LIN {X 0,Y 233.095,Z 584.115,A -85,B 0,C 180,E1 -19797.408,E2 -19797.408} C_VEL
LIN {X 0,Y 233.044,Z 587.862,A -85,B 0,C 180,E1 -19800,E2 -19800} C_VEL
LIN {X 0,Y 233.19,Z 589.815,A -85,B 0,C 180,E1 -19801.727,E2 -19801.727} C_VEL
LIN {X 0,Y 233.829,Z 592.542,A -85,B 0,C 180,E1 -19805.173,E2 -19805.173} C_VEL
LIN {X 0,Y 234.895,Z 593.821,A -85,B 0,C 180,E1 -19808.603,E2 -19808.603} C_VEL
LIN {X 0,Y 236.957,Z 593.579,A -85,B 0,C 180,E1 -19811.982,E2 -19811.982} C_VEL
LIN {X 0,Y 239.578,Z 591.963,A -85,B 0,C 180,E1 -19815.308,E2 -19815.308} C_VEL
LIN {X 0,Y 243.144,Z 588.902,A -85,B 0,C 180,E1 -19818.539,E2 -19818.539} C_VEL
LIN {X 0,Y 247.545,Z 584.286,A -85,B 0,C 180,E1 -19821.659,E2 -19821.659} C_VEL
LIN {X 0,Y 251.345,Z 579.836,A -85,B 0,C 180,E1 -19823.919,E2 -19823.919} C_VEL
LIN {X 0,Y 256.457,Z 573.303,A -85,B 0,C 180,E1 -19826.444,E2 -19826.444} C_VEL
LIN {X 0,Y 262.099,Z 565.298,A -85,B 0,C 180,E1 -19828.859,E2 -19828.859} C_VEL
LIN {X 0,Y 265.58,Z 559.917,A -85,B 0,C 180,E1 -19830.185,E2 -19830.185} C_VEL
LIN {X 0,Y 266.32,Z 558.434,A -85,B 0,C 180,E1 -19830.591,E2 -19830.591} C_VEL
LIN {X 0,Y 266.521,Z 553.535,A -85,B 0,C 180,E1 -19833.039,E2 -19833.039} C_VEL
LIN {X 0,Y 266.277,Z 549.635,A -85,B 0,C 180,E1 -19835.497,E2 -19835.497} C_VEL
LIN {X 0,Y 266.11,Z 548.21,A -85,B 0,C 180,E1 -19836.623,E2 -19836.623} C_VEL
LIN {X 0,Y 265.217,Z 545.882,A -85,B 0,C 180,E1 -19839.783,E2 -19839.783} C_VEL
LIN {X 0,Y 264.843,Z 545.256,A -85,B 0,C 180,E1 -19842.01,E2 -19842.01} C_VEL
LIN {X 0,Y 264.728,Z 545.601,A -85,B 0,C 180,E1 -19844.481,E2 -19844.481} C_VEL
LIN {X 0,Y 264.637,Z 546.784,A -85,B 0,C 180,E1 -19846.331,E2 -19846.331} C_VEL
LIN {X 0,Y 264.615,Z 549.004,A -85,B 0,C 180,E1 -19848.395,E2 -19848.395} C_VEL
LIN {X 0,Y 264.556,Z 552.156,A -85,B 0,C 180,E1 -19850.389,E2 -19850.389} C_VEL
LIN {X 0,Y 264.44,Z 552.98,A -85,B 0,C 180,E1 -19850.801,E2 -19850.801} C_VEL
LIN {X 0,Y 263.759,Z 555.933,A -85,B 0,C 180,E1 -19851.912,E2 -19851.912} C_VEL
LIN {X 0,Y 262.187,Z 559.644,A -85,B 0,C 180,E1 -19852.881,E2 -19852.881} C_VEL
LIN {X 0,Y 257.063,Z 569.958,A -85,B 0,C 180,E1 -19855.355,E2 -19855.355} C_VEL
LIN {X 0,Y 256.138,Z 572.23,A -85,B 0,C 180,E1 -19856.059,E2 -19856.059} C_VEL
LIN {X 0,Y 254.206,Z 577.634,A -85,B 0,C 180,E1 -19857.845,E2 -19857.845} C_VEL
LIN {X 0,Y 251.79,Z 582.561,A -85,B 0,C 180,E1 -19859.376,E2 -19859.376} C_VEL
LIN {X 0,Y 246.124,Z 591,A -85,B 0,C 180,E1 -19861.891,E2 -19861.891} C_VEL
LIN {X 0,Y 240.216,Z 598.91,A -85,B 0,C 180,E1 -19864.898,E2 -19864.898} C_VEL
LIN {X 0,Y 235.324,Z 605.22,A -85,B 0,C 180,E1 -19868.079,E2 -19868.079} C_VEL
LIN {X 0,Y 231.591,Z 610.016,A -85,B 0,C 180,E1 -19871.419,E2 -19871.419} C_VEL
LIN {X 0,Y 229.256,Z 612.702,A -85,B 0,C 180,E1 -19873.984,E2 -19873.984} C_VEL
LIN {X 0,Y 227.193,Z 615.06,A -85,B 0,C 180,E1 -19877.494,E2 -19877.494} C_VEL
LIN {X 0,Y 226.152,Z 616.049,A -85,B 0,C 180,E1 -19881.061,E2 -19881.061} C_VEL
LIN {X 0,Y 225.922,Z 615.639,A -85,B 0,C 180,E1 -19884.645,E2 -19884.645} C_VEL
LIN {X 0,Y 226.286,Z 613.75,A -85,B 0,C 180,E1 -19888.22,E2 -19888.22} C_VEL
LIN {X 0,Y 226.588,Z 612.17,A -85,B 0,C 180,E1 -19890,E2 -19890} C_VEL
LIN {X 0,Y 226.502,Z 608.882,A -85,B 0,C 180,E1 -19892.667,E2 -19892.667} C_VEL
LIN {X 0,Y 226.549,Z 604.491,A -85,B 0,C 180,E1 -19895.34,E2 -19895.34} C_VEL
LIN {X 0,Y 226.752,Z 597.802,A -85,B 0,C 180,E1 -19898.466,E2 -19898.466} C_VEL
LIN {X 0,Y 227.156,Z 590.44,A -85,B 0,C 180,E1 -19901.149,E2 -19901.149} C_VEL
LIN {X 0,Y 227.998,Z 581.33,A -85,B 0,C 180,E1 -19903.821,E2 -19903.821} C_VEL
LIN {X 0,Y 229.113,Z 571.11,A -85,B 0,C 180,E1 -19906.255,E2 -19906.255} C_VEL
LIN {X 0,Y 230.451,Z 559.72,A -85,B 0,C 180,E1 -19908.434,E2 -19908.434} C_VEL
LIN {X 0,Y 229.408,Z 548.685,A -85,B 0,C 180,E1 -19910.16,E2 -19910.16} C_VEL
LIN {X 0,Y 228.165,Z 535.293,A -85,B 0,C 180,E1 -19911.853,E2 -19911.853} C_VEL
LIN {X 0,Y 227.183,Z 521.577,A -85,B 0,C 180,E1 -19913.211,E2 -19913.211} C_VEL
LIN {X 0,Y 226.928,Z 513.581,A -85,B 0,C 180,E1 -19913.863,E2 -19913.863} C_VEL
LIN {X 0,Y 228.074,Z 506.997,A -85,B 0,C 180,E1 -19919.54,E2 -19919.54} C_VEL
LIN {X 0,Y 229.249,Z 501.672,A -85,B 0,C 180,E1 -19924.134,E2 -19924.134} C_VEL
LIN {X 0,Y 229.836,Z 499.05,A -85,B 0,C 180,E1 -19926.414,E2 -19926.414} C_VEL
LIN {X 0,Y 229.367,Z 495.015,A -85,B 0,C 180,E1 -19930.05,E2 -19930.05} C_VEL
LIN {X 0,Y 228.375,Z 489.834,A -85,B 0,C 180,E1 -19934.944,E2 -19934.944} C_VEL
LIN {X 0,Y 228.135,Z 488.069,A -85,B 0,C 180,E1 -19936.73,E2 -19936.73} C_VEL
LIN {X 0,Y 227.881,Z 488.095,A -85,B 0,C 180,E1 -19941.916,E2 -19941.916} C_VEL
LIN {X 0,Y 227.891,Z 488.098,A -85,B 0,C 180,E1 -19946.373,E2 -19946.373} C_VEL
LIN {X 0,Y 227.905,Z 488.095,A -85,B 0,C 180,E1 -19950.436,E2 -19950.436} C_VEL
LIN {X 0,Y 227.929,Z 488.093,A -85,B 0,C 180,E1 -19954.426,E2 -19954.426} C_VEL
LIN {X 0,Y 227.963,Z 488.088,A -85,B 0,C 180,E1 -19958.287,E2 -19958.287} C_VEL
LIN {X 0,Y 228.036,Z 488.08,A -85,B 0,C 180,E1 -19962.826,E2 -19962.826} C_VEL
LIN {X 0,Y 228.095,Z 488.069,A -85,B 0,C 180,E1 -19967.545,E2 -19967.545} C_VEL
LIN {X 0,Y 228.327,Z 488.042,A -85,B 0,C 180,E1 -19971.147,E2 -19971.147} C_VEL
LIN {X 0,Y 228.36,Z 488.039,A -85,B 0,C 180,E1 -19972.929,E2 -19972.929} C_VEL
LIN {X 0,Y 228.556,Z 488.012,A -85,B 0,C 180,E1 -19978.238,E2 -19978.238} C_VEL
LIN {X 0,Y 228.557,Z 488.013,A -85,B 0,C 180,E1 -19981.762,E2 -19981.762} C_VEL
LIN {X 0,Y 228.36,Z 488.036,A -85,B 0,C 180,E1 -19987.072,E2 -19987.072} C_VEL
LIN {X 0,Y 228.173,Z 488.063,A -85,B 0,C 180,E1 -19990.65,E2 -19990.65} C_VEL
LIN {X 0,Y 228.06,Z 488.073,A -85,B 0,C 180,E1 -19996.102,E2 -19996.102} C_VEL
LIN {X 0,Y 227.945,Z 488.09,A -85,B 0,C 180,E1 -19999.826,E2 -19999.826} C_VEL
LIN {X 0,Y 227.916,Z 488.091,A -85,B 0,C 180,E1 -20003.633,E2 -20003.633} C_VEL
LIN {X 0,Y 227.888,Z 488.096,A -85,B 0,C 180,E1 -20007.555,E2 -20007.555} C_VEL
LIN {X 0,Y 227.874,Z 488.097,A -85,B 0,C 180,E1 -20011.622,E2 -20011.622} C_VEL
LIN {X 0,Y 227.885,Z 488.097,A -85,B 0,C 180,E1 -20015.872,E2 -20015.872} C_VEL
LIN {X 0,Y 227.827,Z 488.104,A -85,B 0,C 180,E1 -20020.377,E2 -20020.377} C_VEL
LIN {X 0,Y 227.835,Z 488.103,A -85,B 0,C 180,E1 -20025.193,E2 -20025.193} C_VEL
LIN {X 0,Y 227.835,Z 488.102,A -85,B 0,C 180,E1 -20029.625,E2 -20029.625} C_VEL
LIN {X 0,Y 227.903,Z 488.098,A -85,B 0,C 180,E1 -20034.132,E2 -20034.132} C_VEL
LIN {X 0,Y 227.875,Z 488.097,A -85,B 0,C 180,E1 -20038.379,E2 -20038.379} C_VEL
LIN {X 0,Y 227.888,Z 488.098,A -85,B 0,C 180,E1 -20042.445,E2 -20042.445} C_VEL
LIN {X 0,Y 227.917,Z 488.093,A -85,B 0,C 180,E1 -20046.368,E2 -20046.368} C_VEL
LIN {X 0,Y 227.946,Z 488.092,A -85,B 0,C 180,E1 -20050.175,E2 -20050.175} C_VEL
LIN {X 0,Y 228.061,Z 488.077,A -85,B 0,C 180,E1 -20053.898,E2 -20053.898} C_VEL
LIN {X 0,Y 228.076,Z 488.07,A -85,B 0,C 180,E1 -20057.544,E2 -20057.544} C_VEL
LIN {X 0,Y 228.263,Z 488.05,A -85,B 0,C 180,E1 -20061.145,E2 -20061.145} C_VEL
LIN {X 0,Y 228.315,Z 488.042,A -85,B 0,C 180,E1 -20062.928,E2 -20062.928} C_VEL
LIN {X 0,Y 228.558,Z 488.015,A -85,B 0,C 180,E1 -20068.238,E2 -20068.238} C_VEL
LIN {X 0,Y 228.558,Z 488.015,A -85,B 0,C 180,E1 -20071.762,E2 -20071.762} C_VEL
LIN {X 0,Y 228.328,Z 488.041,A -85,B 0,C 180,E1 -20077.072,E2 -20077.072} C_VEL
LIN {X 0,Y 228.15,Z 488.063,A -85,B 0,C 180,E1 -20080.651,E2 -20080.651} C_VEL
LIN {X 0,Y 228.069,Z 488.074,A -85,B 0,C 180,E1 -20084.272,E2 -20084.272} C_VEL
LIN {X 0,Y 228.007,Z 488.085,A -85,B 0,C 180,E1 -20087.953,E2 -20087.953} C_VEL
LIN {X 0,Y 227.934,Z 488.089,A -85,B 0,C 180,E1 -20092.329,E2 -20092.329} C_VEL
LIN {X 0,Y 227.946,Z 488.089,A -85,B 0,C 180,E1 -20096.603,E2 -20096.603} C_VEL
LIN {X 0,Y 227.911,Z 488.091,A -85,B 0,C 180,E1 -20100.296,E2 -20100.296} C_VEL
LIN {X 0,Y 227.892,Z 488.098,A -85,B 0,C 180,E1 -20103.718,E2 -20103.718} C_VEL
LIN {X 0,Y 227.873,Z 488.098,A -85,B 0,C 180,E1 -20108.086,E2 -20108.086} C_VEL
LIN {X 0,Y 227.817,Z 488.105,A -85,B 0,C 180,E1 -20112.741,E2 -20112.741} C_VEL
LIN {X 0,Y 227.812,Z 488.105,A -85,B 0,C 180,E1 -20117.257,E2 -20117.257} C_VEL
LIN {X 0,Y 227.786,Z 488.112,A -85,B 0,C 180,E1 -20121.897,E2 -20121.897} C_VEL
LIN {X 0,Y 227.697,Z 488.121,A -85,B 0,C 180,E1 -20124.094,E2 -20124.094} C_VEL
LIN {X 0,Y 227.316,Z 488.167,A -85,B 0,C 180,E1 -20128.291,E2 -20128.291} C_VEL
LIN {X 0,Y 226.929,Z 488.222,A -85,B 0,C 180,E1 -20132.318,E2 -20132.318} C_VEL
LIN {X 0,Y 226.517,Z 488.272,A -85,B 0,C 180,E1 -20136.502,E2 -20136.502} C_VEL
LIN {X 0,Y 229.096,Z 503.824,A -85,B 0,C 180,E1 -20137.96,E2 -20137.96} C_VEL
LIN {X 0,Y 231.348,Z 516.521,A -85,B 0,C 180,E1 -20139.475,E2 -20139.475} C_VEL
LIN {X 0,Y 232.042,Z 520.942,A -85,B 0,C 180,E1 -20140.077,E2 -20140.077} C_VEL
LIN {X 0,Y 230.695,Z 533.731,A -85,B 0,C 180,E1 -20142.034,E2 -20142.034} C_VEL
LIN {X 0,Y 229.335,Z 545.229,A -85,B 0,C 180,E1 -20144.218,E2 -20144.218} C_VEL
LIN {X 0,Y 228.115,Z 555.573,A -85,B 0,C 180,E1 -20146.64,E2 -20146.64} C_VEL
LIN {X 0,Y 227.179,Z 564.818,A -85,B 0,C 180,E1 -20149.303,E2 -20149.303} C_VEL
LIN {X 0,Y 226.466,Z 573.528,A -85,B 0,C 180,E1 -20152.421,E2 -20152.421} C_VEL
LIN {X 0,Y 226.079,Z 580.412,A -85,B 0,C 180,E1 -20155.542,E2 -20155.542} C_VEL
LIN {X 0,Y 225.985,Z 585.073,A -85,B 0,C 180,E1 -20158.218,E2 -20158.218} C_VEL
LIN {X 0,Y 226.119,Z 589.684,A -85,B 0,C 180,E1 -20161.781,E2 -20161.781} C_VEL
LIN {X 0,Y 226.405,Z 591.403,A -85,B 0,C 180,E1 -20163.559,E2 -20163.559} C_VEL
LIN {X 0,Y 227.226,Z 593.653,A -85,B 0,C 180,E1 -20167.106,E2 -20167.106} C_VEL
LIN {X 0,Y 228.857,Z 594.476,A -85,B 0,C 180,E1 -20170.617,E2 -20170.617} C_VEL
LIN {X 0,Y 231.32,Z 593.867,A -85,B 0,C 180,E1 -20174.067,E2 -20174.067} C_VEL
LIN {X 0,Y 234.616,Z 591.845,A -85,B 0,C 180,E1 -20177.431,E2 -20177.431} C_VEL
LIN {X 0,Y 238.783,Z 588.417,A -85,B 0,C 180,E1 -20180.682,E2 -20180.682} C_VEL
LIN {X 0,Y 243.747,Z 583.472,A -85,B 0,C 180,E1 -20183.807,E2 -20183.807} C_VEL
LIN {X 0,Y 249.667,Z 576.905,A -85,B 0,C 180,E1 -20186.769,E2 -20186.769} C_VEL
LIN {X 0,Y 256.354,Z 568.409,A -85,B 0,C 180,E1 -20189.569,E2 -20189.569} C_VEL
LIN {X 0,Y 259.937,Z 563.469,A -85,B 0,C 180,E1 -20190.911,E2 -20190.911} C_VEL
LIN {X 0,Y 261.012,Z 561.597,A -85,B 0,C 180,E1 -20191.474,E2 -20191.474} C_VEL
LIN {X 0,Y 261.39,Z 557.918,A -85,B 0,C 180,E1 -20193.54,E2 -20193.54} C_VEL
LIN {X 0,Y 261.426,Z 554.117,A -85,B 0,C 180,E1 -20196.244,E2 -20196.244} C_VEL
LIN {X 0,Y 260.976,Z 552.102,A -85,B 0,C 180,E1 -20198.651,E2 -20198.651} C_VEL
LIN {X 0,Y 260.607,Z 551.108,A -85,B 0,C 180,E1 -20200.965,E2 -20200.965} C_VEL
LIN {X 0,Y 260.477,Z 550.912,A -85,B 0,C 180,E1 -20203.239,E2 -20203.239} C_VEL
LIN {X 0,Y 260.343,Z 551.8,A -85,B 0,C 180,E1 -20205.422,E2 -20205.422} C_VEL
LIN {X 0,Y 260.165,Z 553.684,A -85,B 0,C 180,E1 -20207.519,E2 -20207.519} C_VEL
LIN {X 0,Y 259.949,Z 556.429,A -85,B 0,C 180,E1 -20209.544,E2 -20209.544} C_VEL
LIN {X 0,Y 259.251,Z 560.111,A -85,B 0,C 180,E1 -20211.427,E2 -20211.427} C_VEL
LIN {X 0,Y 257.672,Z 566.9,A -85,B 0,C 180,E1 -20214.152,E2 -20214.152} C_VEL
LIN {X 0,Y 256.138,Z 572.23,A -85,B 0,C 180,E1 -20216.059,E2 -20216.059} C_VEL
LIN {X 0,Y 255.085,Z 574.558,A -85,B 0,C 180,E1 -20216.743,E2 -20216.743} C_VEL
LIN {X 0,Y 253.54,Z 577.077,A -85,B 0,C 180,E1 -20217.348,E2 -20217.348} C_VEL
LIN {X 0,Y 249.505,Z 582.161,A -85,B 0,C 180,E1 -20218.416,E2 -20218.416} C_VEL
LIN {X 0,Y 242.787,Z 589.348,A -85,B 0,C 180,E1 -20220.062,E2 -20220.062} C_VEL
LIN {X 0,Y 240.884,Z 591.498,A -85,B 0,C 180,E1 -20220.727,E2 -20220.727} C_VEL
LIN {X 0,Y 235.306,Z 598.328,A -85,B 0,C 180,E1 -20223.383,E2 -20223.383} C_VEL
LIN {X 0,Y 229.312,Z 605.282,A -85,B 0,C 180,E1 -20227.027,E2 -20227.027} C_VEL
LIN {X 0,Y 225.718,Z 609.319,A -85,B 0,C 180,E1 -20229.971,E2 -20229.971} C_VEL
LIN {X 0,Y 222.436,Z 612.714,A -85,B 0,C 180,E1 -20233.479,E2 -20233.479} C_VEL
LIN {X 0,Y 220.225,Z 614.779,A -85,B 0,C 180,E1 -20237.092,E2 -20237.092} C_VEL
LIN {X 0,Y 219.122,Z 615.507,A -85,B 0,C 180,E1 -20240.772,E2 -20240.772} C_VEL
LIN {X 0,Y 218.886,Z 614.813,A -85,B 0,C 180,E1 -20244.472,E2 -20244.472} C_VEL
LIN {X 0,Y 219.274,Z 612.657,A -85,B 0,C 180,E1 -20248.163,E2 -20248.163} C_VEL
LIN {X 0,Y 219.571,Z 610.998,A -85,B 0,C 180,E1 -20250,E2 -20250} C_VEL
LIN {X 0,Y 219.498,Z 607.509,A -85,B 0,C 180,E1 -20252.753,E2 -20252.753} C_VEL
LIN {X 0,Y 219.557,Z 602.876,A -85,B 0,C 180,E1 -20255.51,E2 -20255.51} C_VEL
LIN {X 0,Y 219.734,Z 596.979,A -85,B 0,C 180,E1 -20258.275,E2 -20258.275} C_VEL
LIN {X 0,Y 220.121,Z 589.583,A -85,B 0,C 180,E1 -20261.044,E2 -20261.044} C_VEL
LIN {X 0,Y 220.962,Z 580.515,A -85,B 0,C 180,E1 -20263.801,E2 -20263.801} C_VEL
LIN {X 0,Y 221.952,Z 571.302,A -85,B 0,C 180,E1 -20266.085,E2 -20266.085} C_VEL
LIN {X 0,Y 223.289,Z 560.005,A -85,B 0,C 180,E1 -20268.346,E2 -20268.346} C_VEL
LIN {X 0,Y 222.297,Z 548.841,A -85,B 0,C 180,E1 -20270.17,E2 -20270.17} C_VEL
LIN {X 0,Y 221.092,Z 535.554,A -85,B 0,C 180,E1 -20271.932,E2 -20271.932} C_VEL
LIN {X 0,Y 220.099,Z 521.557,A -85,B 0,C 180,E1 -20273.386,E2 -20273.386} C_VEL
LIN {X 0,Y 219.834,Z 513.247,A -85,B 0,C 180,E1 -20274.054,E2 -20274.054} C_VEL
LIN {X 0,Y 220.969,Z 507.128,A -85,B 0,C 180,E1 -20279.537,E2 -20279.537} C_VEL
LIN {X 0,Y 222.295,Z 501.353,A -85,B 0,C 180,E1 -20284.714,E2 -20284.714} C_VEL
LIN {X 0,Y 222.721,Z 498.997,A -85,B 0,C 180,E1 -20286.837,E2 -20286.837} C_VEL
LIN {X 0,Y 222.163,Z 495.001,A -85,B 0,C 180,E1 -20290.604,E2 -20290.604} C_VEL
LIN {X 0,Y 221.201,Z 489.839,A -85,B 0,C 180,E1 -20295.655,E2 -20295.655} C_VEL
LIN {X 0,Y 221.104,Z 488.945,A -85,B 0,C 180,E1 -20296.774,E2 -20296.774} C_VEL
LIN {X 0,Y 220.866,Z 488.973,A -85,B 0,C 180,E1 -20300.476,E2 -20300.476} C_VEL
LIN {X 0,Y 220.816,Z 488.979,A -85,B 0,C 180,E1 -20305.048,E2 -20305.048} C_VEL
LIN {X 0,Y 220.834,Z 488.974,A -85,B 0,C 180,E1 -20309.39,E2 -20309.39} C_VEL
LIN {X 0,Y 220.895,Z 488.966,A -85,B 0,C 180,E1 -20313.55,E2 -20313.55} C_VEL
LIN {X 0,Y 220.879,Z 488.969,A -85,B 0,C 180,E1 -20317.554,E2 -20317.554} C_VEL
LIN {X 0,Y 220.985,Z 488.958,A -85,B 0,C 180,E1 -20322.571,E2 -20322.571} C_VEL
LIN {X 0,Y 221.028,Z 488.95,A -85,B 0,C 180,E1 -20327.14,E2 -20327.14} C_VEL
LIN {X 0,Y 221.26,Z 488.923,A -85,B 0,C 180,E1 -20330.862,E2 -20330.862} C_VEL
LIN {X 0,Y 221.313,Z 488.918,A -85,B 0,C 180,E1 -20332.703,E2 -20332.703} C_VEL
LIN {X 0,Y 221.514,Z 488.889,A -85,B 0,C 180,E1 -20338.182,E2 -20338.182} C_VEL
LIN {X 0,Y 221.515,Z 488.891,A -85,B 0,C 180,E1 -20341.818,E2 -20341.818} C_VEL
LIN {X 0,Y 221.313,Z 488.913,A -85,B 0,C 180,E1 -20347.298,E2 -20347.298} C_VEL
LIN {X 0,Y 221.119,Z 488.94,A -85,B 0,C 180,E1 -20350.994,E2 -20350.994} C_VEL
LIN {X 0,Y 221.018,Z 488.953,A -85,B 0,C 180,E1 -20356.63,E2 -20356.63} C_VEL
LIN {X 0,Y 220.895,Z 488.97,A -85,B 0,C 180,E1 -20360.486,E2 -20360.486} C_VEL
LIN {X 0,Y 220.869,Z 488.971,A -85,B 0,C 180,E1 -20364.435,E2 -20364.435} C_VEL
LIN {X 0,Y 220.839,Z 488.977,A -85,B 0,C 180,E1 -20368.514,E2 -20368.514} C_VEL
LIN {X 0,Y 220.822,Z 488.974,A -85,B 0,C 180,E1 -20372.756,E2 -20372.756} C_VEL
LIN {X 0,Y 220.813,Z 488.978,A -85,B 0,C 180,E1 -20377.279,E2 -20377.279} C_VEL
LIN {X 0,Y 220.772,Z 488.981,A -85,B 0,C 180,E1 -20381.953,E2 -20381.953} C_VEL
LIN {X 0,Y 220.776,Z 488.982,A -85,B 0,C 180,E1 -20385.547,E2 -20385.547} C_VEL
LIN {X 0,Y 220.812,Z 488.977,A -85,B 0,C 180,E1 -20390.464,E2 -20390.464} C_VEL
LIN {X 0,Y 220.834,Z 488.975,A -85,B 0,C 180,E1 -20392.795,E2 -20392.795} C_VEL
LIN {X 0,Y 220.827,Z 488.975,A -85,B 0,C 180,E1 -20397.246,E2 -20397.246} C_VEL
LIN {X 0,Y 220.839,Z 488.974,A -85,B 0,C 180,E1 -20401.487,E2 -20401.487} C_VEL
LIN {X 0,Y 220.87,Z 488.971,A -85,B 0,C 180,E1 -20405.566,E2 -20405.566} C_VEL
LIN {X 0,Y 220.896,Z 488.966,A -85,B 0,C 180,E1 -20409.514,E2 -20409.514} C_VEL
LIN {X 0,Y 221.02,Z 488.952,A -85,B 0,C 180,E1 -20413.371,E2 -20413.371} C_VEL
LIN {X 0,Y 221.085,Z 488.943,A -85,B 0,C 180,E1 -20419.005,E2 -20419.005} C_VEL
LIN {X 0,Y 221.252,Z 488.923,A -85,B 0,C 180,E1 -20422.701,E2 -20422.701} C_VEL
LIN {X 0,Y 221.515,Z 488.893,A -85,B 0,C 180,E1 -20428.182,E2 -20428.182} C_VEL
LIN {X 0,Y 221.516,Z 488.893,A -85,B 0,C 180,E1 -20431.818,E2 -20431.818} C_VEL
LIN {X 0,Y 221.263,Z 488.921,A -85,B 0,C 180,E1 -20437.3,E2 -20437.3} C_VEL
LIN {X 0,Y 221.086,Z 488.943,A -85,B 0,C 180,E1 -20440.996,E2 -20440.996} C_VEL
LIN {X 0,Y 221.021,Z 488.952,A -85,B 0,C 180,E1 -20446.63,E2 -20446.63} C_VEL
LIN {X 0,Y 220.897,Z 488.966,A -85,B 0,C 180,E1 -20450.486,E2 -20450.486} C_VEL
LIN {X 0,Y 220.871,Z 488.971,A -85,B 0,C 180,E1 -20454.435,E2 -20454.435} C_VEL
LIN {X 0,Y 220.84,Z 488.973,A -85,B 0,C 180,E1 -20458.513,E2 -20458.513} C_VEL
LIN {X 0,Y 220.827,Z 488.975,A -85,B 0,C 180,E1 -20462.755,E2 -20462.755} C_VEL
LIN {X 0,Y 220.842,Z 488.974,A -85,B 0,C 180,E1 -20467.288,E2 -20467.288} C_VEL
LIN {X 0,Y 220.778,Z 488.984,A -85,B 0,C 180,E1 -20471.951,E2 -20471.951} C_VEL
LIN {X 0,Y 220.776,Z 488.985,A -85,B 0,C 180,E1 -20475.546,E2 -20475.546} C_VEL
LIN {X 0,Y 220.771,Z 488.982,A -85,B 0,C 180,E1 -20480.455,E2 -20480.455} C_VEL
LIN {X 0,Y 220.718,Z 488.99,A -85,B 0,C 180,E1 -20482.771,E2 -20482.771} C_VEL
LIN {X 0,Y 220.364,Z 489.031,A -85,B 0,C 180,E1 -20487.167,E2 -20487.167} C_VEL
LIN {X 0,Y 219.979,Z 489.083,A -85,B 0,C 180,E1 -20491.365,E2 -20491.365} C_VEL
LIN {X 0,Y 219.534,Z 489.276,A -85,B 0,C 180,E1 -20496.349,E2 -20496.349} C_VEL
LIN {X 0,Y 221.785,Z 503.009,A -85,B 0,C 180,E1 -20497.65,E2 -20497.65} C_VEL
LIN {X 0,Y 224.089,Z 516.032,A -85,B 0,C 180,E1 -20499.22,E2 -20499.22} C_VEL
LIN {X 0,Y 224.938,Z 520.869,A -85,B 0,C 180,E1 -20499.898,E2 -20499.898} C_VEL
LIN {X 0,Y 223.614,Z 533.665,A -85,B 0,C 180,E1 -20501.918,E2 -20501.918} C_VEL
LIN {X 0,Y 222.223,Z 545.155,A -85,B 0,C 180,E1 -20504.17,E2 -20504.17} C_VEL
LIN {X 0,Y 221.006,Z 555.514,A -85,B 0,C 180,E1 -20506.67,E2 -20506.67} C_VEL
LIN {X 0,Y 220.071,Z 564.873,A -85,B 0,C 180,E1 -20509.419,E2 -20509.419} C_VEL
LIN {X 0,Y 219.346,Z 573.658,A -85,B 0,C 180,E1 -20512.636,E2 -20512.636} C_VEL
LIN {X 0,Y 219.007,Z 579.696,A -85,B 0,C 180,E1 -20515.398,E2 -20515.398} C_VEL
LIN {X 0,Y 218.919,Z 584.567,A -85,B 0,C 180,E1 -20518.16,E2 -20518.16} C_VEL
LIN {X 0,Y 218.945,Z 588.414,A -85,B 0,C 180,E1 -20520.919,E2 -20520.919} C_VEL
LIN {X 0,Y 219.346,Z 591.333,A -85,B 0,C 180,E1 -20523.674,E2 -20523.674} C_VEL
LIN {X 0,Y 220.182,Z 593.907,A -85,B 0,C 180,E1 -20527.335,E2 -20527.335} C_VEL
LIN {X 0,Y 221.913,Z 595.009,A -85,B 0,C 180,E1 -20530.954,E2 -20530.954} C_VEL
LIN {X 0,Y 224.511,Z 594.714,A -85,B 0,C 180,E1 -20534.503,E2 -20534.503} C_VEL
LIN {X 0,Y 227.955,Z 593.059,A -85,B 0,C 180,E1 -20537.957,E2 -20537.957} C_VEL
LIN {X 0,Y 232.315,Z 589.99,A -85,B 0,C 180,E1 -20541.286,E2 -20541.286} C_VEL
LIN {X 0,Y 237.53,Z 585.478,A -85,B 0,C 180,E1 -20544.471,E2 -20544.471} C_VEL
LIN {X 0,Y 242.051,Z 581.058,A -85,B 0,C 180,E1 -20546.746,E2 -20546.746} C_VEL
LIN {X 0,Y 248.862,Z 573.648,A -85,B 0,C 180,E1 -20549.618,E2 -20549.618} C_VEL
LIN {X 0,Y 255.215,Z 565.676,A -85,B 0,C 180,E1 -20552.002,E2 -20552.002} C_VEL
LIN {X 0,Y 255.674,Z 564.787,A -85,B 0,C 180,E1 -20552.393,E2 -20552.393} C_VEL
LIN {X 0,Y 256.29,Z 560.636,A -85,B 0,C 180,E1 -20555.16,E2 -20555.16} C_VEL
LIN {X 0,Y 256.446,Z 559.334,A -85,B 0,C 180,E1 -20556.23,E2 -20556.23} C_VEL
LIN {X 0,Y 256.152,Z 557.161,A -85,B 0,C 180,E1 -20559.127,E2 -20559.127} C_VEL
LIN {X 0,Y 255.896,Z 556.341,A -85,B 0,C 180,E1 -20562.137,E2 -20562.137} C_VEL
LIN {X 0,Y 255.815,Z 556.712,A -85,B 0,C 180,E1 -20564.414,E2 -20564.414} C_VEL
LIN {X 0,Y 255.553,Z 558.206,A -85,B 0,C 180,E1 -20566.565,E2 -20566.565} C_VEL
LIN {X 0,Y 255.244,Z 560.565,A -85,B 0,C 180,E1 -20568.637,E2 -20568.637} C_VEL
LIN {X 0,Y 254.383,Z 564.117,A -85,B 0,C 180,E1 -20570.676,E2 -20570.676} C_VEL
LIN {X 0,Y 252.559,Z 570.004,A -85,B 0,C 180,E1 -20573.254,E2 -20573.254} C_VEL
LIN {X 0,Y 250.113,Z 576.663,A -85,B 0,C 180,E1 -20575.806,E2 -20575.806} C_VEL
LIN {X 0,Y 247.423,Z 582.413,A -85,B 0,C 180,E1 -20577.819,E2 -20577.819} C_VEL
LIN {X 0,Y 244.311,Z 587.131,A -85,B 0,C 180,E1 -20579.295,E2 -20579.295} C_VEL
LIN {X 0,Y 240.884,Z 591.498,A -85,B 0,C 180,E1 -20580.727,E2 -20580.727} C_VEL
LIN {X 0,Y 237.881,Z 594.617,A -85,B 0,C 180,E1 -20581.71,E2 -20581.71} C_VEL
LIN {X 0,Y 231.696,Z 599.436,A -85,B 0,C 180,E1 -20583.21,E2 -20583.21} C_VEL
LIN {X 0,Y 225.744,Z 603.53,A -85,B 0,C 180,E1 -20584.876,E2 -20584.876} C_VEL
LIN {X 0,Y 223.156,Z 605.615,A -85,B 0,C 180,E1 -20586.101,E2 -20586.101} C_VEL
LIN {X 0,Y 219.064,Z 609.662,A -85,B 0,C 180,E1 -20589.335,E2 -20589.335} C_VEL
LIN {X 0,Y 215.637,Z 612.711,A -85,B 0,C 180,E1 -20592.943,E2 -20592.943} C_VEL
LIN {X 0,Y 213.273,Z 614.435,A -85,B 0,C 180,E1 -20596.663,E2 -20596.663} C_VEL
LIN {X 0,Y 212.11,Z 614.85,A -85,B 0,C 180,E1 -20600.464,E2 -20600.464} C_VEL
LIN {X 0,Y 211.851,Z 613.876,A -85,B 0,C 180,E1 -20604.401,E2 -20604.401} C_VEL
LIN {X 0,Y 212.259,Z 611.533,A -85,B 0,C 180,E1 -20608.102,E2 -20608.102} C_VEL
LIN {X 0,Y 212.573,Z 608.615,A -85,B 0,C 180,E1 -20610.947,E2 -20610.947} C_VEL
LIN {X 0,Y 212.531,Z 604.553,A -85,B 0,C 180,E1 -20613.792,E2 -20613.792} C_VEL
LIN {X 0,Y 212.622,Z 599.223,A -85,B 0,C 180,E1 -20616.68,E2 -20616.68} C_VEL
LIN {X 0,Y 212.869,Z 592.598,A -85,B 0,C 180,E1 -20619.502,E2 -20619.502} C_VEL
LIN {X 0,Y 213.534,Z 584.346,A -85,B 0,C 180,E1 -20622.353,E2 -20622.353} C_VEL
LIN {X 0,Y 214.326,Z 576.01,A -85,B 0,C 180,E1 -20624.722,E2 -20624.722} C_VEL
LIN {X 0,Y 215.422,Z 566.005,A -85,B 0,C 180,E1 -20627.075,E2 -20627.075} C_VEL
LIN {X 0,Y 216.192,Z 558.913,A -85,B 0,C 180,E1 -20628.479,E2 -20628.479} C_VEL
LIN {X 0,Y 215.083,Z 547.939,A -85,B 0,C 180,E1 -20630.318,E2 -20630.318} C_VEL
LIN {X 0,Y 213.908,Z 534.706,A -85,B 0,C 180,E1 -20632.118,E2 -20632.118} C_VEL
LIN {X 0,Y 213.011,Z 521.041,A -85,B 0,C 180,E1 -20633.581,E2 -20633.581} C_VEL
LIN {X 0,Y 212.774,Z 512.815,A -85,B 0,C 180,E1 -20634.321,E2 -20634.321} C_VEL
LIN {X 0,Y 213.853,Z 507.235,A -85,B 0,C 180,E1 -20639.535,E2 -20639.535} C_VEL
LIN {X 0,Y 214.922,Z 502.687,A -85,B 0,C 180,E1 -20643.773,E2 -20643.773} C_VEL
LIN {X 0,Y 215.537,Z 500.368,A -85,B 0,C 180,E1 -20645.939,E2 -20645.939} C_VEL
LIN {X 0,Y 215.47,Z 497.696,A -85,B 0,C 180,E1 -20648.482,E2 -20648.482} C_VEL
LIN {X 0,Y 214.701,Z 493.695,A -85,B 0,C 180,E1 -20652.439,E2 -20652.439} C_VEL
LIN {X 0,Y 214.068,Z 489.821,A -85,B 0,C 180,E1 -20656.576,E2 -20656.576} C_VEL
LIN {X 0,Y 213.785,Z 489.851,A -85,B 0,C 180,E1 -20662.09,E2 -20662.09} C_VEL
LIN {X 0,Y 213.77,Z 489.855,A -85,B 0,C 180,E1 -20666.02,E2 -20666.02} C_VEL
LIN {X 0,Y 213.761,Z 489.857,A -85,B 0,C 180,E1 -20670.451,E2 -20670.451} C_VEL
LIN {X 0,Y 213.802,Z 489.854,A -85,B 0,C 180,E1 -20674.702,E2 -20674.702} C_VEL
LIN {X 0,Y 213.814,Z 489.849,A -85,B 0,C 180,E1 -20678.804,E2 -20678.804} C_VEL
LIN {X 0,Y 213.945,Z 489.836,A -85,B 0,C 180,E1 -20682.804,E2 -20682.804} C_VEL
LIN {X 0,Y 213.982,Z 489.83,A -85,B 0,C 180,E1 -20686.709,E2 -20686.709} C_VEL
LIN {X 0,Y 214.198,Z 489.802,A -85,B 0,C 180,E1 -20690.558,E2 -20690.558} C_VEL
LIN {X 0,Y 214.25,Z 489.798,A -85,B 0,C 180,E1 -20692.461,E2 -20692.461} C_VEL
LIN {X 0,Y 214.448,Z 489.768,A -85,B 0,C 180,E1 -20698.122,E2 -20698.122} C_VEL
LIN {X 0,Y 214.552,Z 489.757,A -85,B 0,C 180,E1 -20700,E2 -20700} C_VEL
LIN {X 0,Y 214.448,Z 489.771,A -85,B 0,C 180,E1 -20701.878,E2 -20701.878} C_VEL
LIN {X 0,Y 214.25,Z 489.793,A -85,B 0,C 180,E1 -20707.54,E2 -20707.54} C_VEL
LIN {X 0,Y 214.049,Z 489.82,A -85,B 0,C 180,E1 -20711.362,E2 -20711.362} C_VEL
LIN {X 0,Y 213.935,Z 489.83,A -85,B 0,C 180,E1 -20715.237,E2 -20715.237} C_VEL
LIN {X 0,Y 213.842,Z 489.846,A -85,B 0,C 180,E1 -20719.188,E2 -20719.188} C_VEL
LIN {X 0,Y 213.849,Z 489.842,A -85,B 0,C 180,E1 -20723.227,E2 -20723.227} C_VEL
LIN {X 0,Y 213.831,Z 489.847,A -85,B 0,C 180,E1 -20727.45,E2 -20727.45} C_VEL
LIN {X 0,Y 213.78,Z 489.853,A -85,B 0,C 180,E1 -20731.736,E2 -20731.736} C_VEL
LIN {X 0,Y 213.746,Z 489.861,A -85,B 0,C 180,E1 -20736.288,E2 -20736.288} C_VEL
LIN {X 0,Y 213.714,Z 489.859,A -85,B 0,C 180,E1 -20741.126,E2 -20741.126} C_VEL
LIN {X 0,Y 213.708,Z 489.862,A -85,B 0,C 180,E1 -20743.679,E2 -20743.679} C_VEL
LIN {X 0,Y 213.71,Z 489.866,A -85,B 0,C 180,E1 -20746.344,E2 -20746.344} C_VEL
LIN {X 0,Y 213.738,Z 489.856,A -85,B 0,C 180,E1 -20751.337,E2 -20751.337} C_VEL
LIN {X 0,Y 213.773,Z 489.857,A -85,B 0,C 180,E1 -20756.021,E2 -20756.021} C_VEL
LIN {X 0,Y 213.783,Z 489.854,A -85,B 0,C 180,E1 -20760.455,E2 -20760.455} C_VEL
LIN {X 0,Y 213.805,Z 489.851,A -85,B 0,C 180,E1 -20764.702,E2 -20764.702} C_VEL
LIN {X 0,Y 213.817,Z 489.847,A -85,B 0,C 180,E1 -20768.804,E2 -20768.804} C_VEL
LIN {X 0,Y 213.947,Z 489.833,A -85,B 0,C 180,E1 -20772.804,E2 -20772.804} C_VEL
LIN {X 0,Y 213.957,Z 489.828,A -85,B 0,C 180,E1 -20776.707,E2 -20776.707} C_VEL
LIN {X 0,Y 214.14,Z 489.81,A -85,B 0,C 180,E1 -20780.555,E2 -20780.555} C_VEL
LIN {X 0,Y 214.095,Z 489.813,A -85,B 0,C 180,E1 -20784.349,E2 -20784.349} C_VEL
LIN {X 0,Y 214.448,Z 489.773,A -85,B 0,C 180,E1 -20788.122,E2 -20788.122} C_VEL
LIN {X 0,Y 214.554,Z 489.761,A -85,B 0,C 180,E1 -20790,E2 -20790} C_VEL
LIN {X 0,Y 214.449,Z 489.773,A -85,B 0,C 180,E1 -20791.878,E2 -20791.878} C_VEL
LIN {X 0,Y 214.203,Z 489.802,A -85,B 0,C 180,E1 -20797.542,E2 -20797.542} C_VEL
LIN {X 0,Y 214.012,Z 489.825,A -85,B 0,C 180,E1 -20801.364,E2 -20801.364} C_VEL
LIN {X 0,Y 213.938,Z 489.833,A -85,B 0,C 180,E1 -20805.237,E2 -20805.237} C_VEL
LIN {X 0,Y 213.844,Z 489.846,A -85,B 0,C 180,E1 -20809.187,E2 -20809.187} C_VEL
LIN {X 0,Y 213.851,Z 489.843,A -85,B 0,C 180,E1 -20813.227,E2 -20813.227} C_VEL
LIN {X 0,Y 213.832,Z 489.849,A -85,B 0,C 180,E1 -20817.45,E2 -20817.45} C_VEL
LIN {X 0,Y 213.782,Z 489.853,A -85,B 0,C 180,E1 -20821.735,E2 -20821.735} C_VEL
LIN {X 0,Y 213.755,Z 489.857,A -85,B 0,C 180,E1 -20826.286,E2 -20826.286} C_VEL
LIN {X 0,Y 213.719,Z 489.86,A -85,B 0,C 180,E1 -20831.124,E2 -20831.124} C_VEL
LIN {X 0,Y 213.711,Z 489.866,A -85,B 0,C 180,E1 -20833.678,E2 -20833.678} C_VEL
LIN {X 0,Y 213.707,Z 489.862,A -85,B 0,C 180,E1 -20836.344,E2 -20836.344} C_VEL
LIN {X 0,Y 213.709,Z 489.86,A -85,B 0,C 180,E1 -20839.146,E2 -20839.146} C_VEL
LIN {X 0,Y 213.582,Z 489.882,A -85,B 0,C 180,E1 -20843.679,E2 -20843.679} C_VEL
LIN {X 0,Y 213.468,Z 489.891,A -85,B 0,C 180,E1 -20845.965,E2 -20845.965} C_VEL
LIN {X 0,Y 213.018,Z 489.949,A -85,B 0,C 180,E1 -20850.337,E2 -20850.337} C_VEL
LIN {X 0,Y 212.515,Z 490.014,A -85,B 0,C 180,E1 -20855.582,E2 -20855.582} C_VEL
LIN {X 0,Y 212.5,Z 490.146,A -85,B 0,C 180,E1 -20856.196,E2 -20856.196} C_VEL
LIN {X 0,Y 214.647,Z 503.47,A -85,B 0,C 180,E1 -20857.515,E2 -20857.515} C_VEL
LIN {X 0,Y 216.917,Z 516.36,A -85,B 0,C 180,E1 -20859.121,E2 -20859.121} C_VEL
LIN {X 0,Y 217.813,Z 521.699,A -85,B 0,C 180,E1 -20859.892,E2 -20859.892} C_VEL
LIN {X 0,Y 216.34,Z 534.619,A -85,B 0,C 180,E1 -20862.024,E2 -20862.024} C_VEL
LIN {X 0,Y 214.988,Z 546.01,A -85,B 0,C 180,E1 -20864.354,E2 -20864.354} C_VEL
LIN {X 0,Y 213.744,Z 557.187,A -85,B 0,C 180,E1 -20867.176,E2 -20867.176} C_VEL
LIN {X 0,Y 212.781,Z 566.237,A -85,B 0,C 180,E1 -20870.014,E2 -20870.014} C_VEL
LIN {X 0,Y 212.223,Z 573.67,A -85,B 0,C 180,E1 -20872.866,E2 -20872.866} C_VEL
LIN {X 0,Y 211.878,Z 580.7,A -85,B 0,C 180,E1 -20876.196,E2 -20876.196} C_VEL
LIN {X 0,Y 211.813,Z 585.479,A -85,B 0,C 180,E1 -20879.049,E2 -20879.049} C_VEL
LIN {X 0,Y 211.983,Z 589.213,A -85,B 0,C 180,E1 -20881.9,E2 -20881.9} C_VEL
LIN {X 0,Y 212.268,Z 591.211,A -85,B 0,C 180,E1 -20883.796,E2 -20883.796} C_VEL
LIN {X 0,Y 213.144,Z 594.049,A -85,B 0,C 180,E1 -20887.579,E2 -20887.579} C_VEL
LIN {X 0,Y 214.98,Z 595.485,A -85,B 0,C 180,E1 -20891.312,E2 -20891.312} C_VEL
LIN {X 0,Y 217.694,Z 595.53,A -85,B 0,C 180,E1 -20894.967,E2 -20894.967} C_VEL
LIN {X 0,Y 221.307,Z 594.2,A -85,B 0,C 180,E1 -20898.516,E2 -20898.516} C_VEL
LIN {X 0,Y 225.874,Z 591.51,A -85,B 0,C 180,E1 -20901.924,E2 -20901.924} C_VEL
LIN {X 0,Y 231.328,Z 587.444,A -85,B 0,C 180,E1 -20905.172,E2 -20905.172} C_VEL
LIN {X 0,Y 237.705,Z 581.827,A -85,B 0,C 180,E1 -20908.233,E2 -20908.233} C_VEL
LIN {X 0,Y 243.109,Z 576.495,A -85,B 0,C 180,E1 -20910.391,E2 -20910.391} C_VEL
LIN {X 0,Y 249.815,Z 569.111,A -85,B 0,C 180,E1 -20912.79,E2 -20912.79} C_VEL
LIN {X 0,Y 250.286,Z 568.244,A -85,B 0,C 180,E1 -20913.2,E2 -20913.2} C_VEL
LIN {X 0,Y 251.094,Z 564.9,A -85,B 0,C 180,E1 -20915.737,E2 -20915.737} C_VEL
LIN {X 0,Y 251.194,Z 562.72,A -85,B 0,C 180,E1 -20918.427,E2 -20918.427} C_VEL
LIN {X 0,Y 251.132,Z 561.727,A -85,B 0,C 180,E1 -20920.921,E2 -20920.921} C_VEL
LIN {X 0,Y 251.132,Z 561.648,A -85,B 0,C 180,E1 -20923.312,E2 -20923.312} C_VEL
LIN {X 0,Y 250.88,Z 562.7,A -85,B 0,C 180,E1 -20925.546,E2 -20925.546} C_VEL
LIN {X 0,Y 250.468,Z 564.633,A -85,B 0,C 180,E1 -20927.667,E2 -20927.667} C_VEL
LIN {X 0,Y 249.603,Z 567.498,A -85,B 0,C 180,E1 -20929.638,E2 -20929.638} C_VEL
LIN {X 0,Y 247.414,Z 573.119,A -85,B 0,C 180,E1 -20932.359,E2 -20932.359} C_VEL
LIN {X 0,Y 244.662,Z 579.291,A -85,B 0,C 180,E1 -20934.935,E2 -20934.935} C_VEL
LIN {X 0,Y 242.393,Z 583.569,A -85,B 0,C 180,E1 -20936.572,E2 -20936.572} C_VEL
LIN {X 0,Y 240.177,Z 586.834,A -85,B 0,C 180,E1 -20937.722,E2 -20937.722} C_VEL
LIN {X 0,Y 233.974,Z 594.177,A -85,B 0,C 180,E1 -20940.289,E2 -20940.289} C_VEL
LIN {X 0,Y 227.589,Z 601.098,A -85,B 0,C 180,E1 -20943.399,E2 -20943.399} C_VEL
LIN {X 0,Y 223.156,Z 605.615,A -85,B 0,C 180,E1 -20946.101,E2 -20946.101} C_VEL
LIN {X 0,Y 220.658,Z 607.548,A -85,B 0,C 180,E1 -20947.397,E2 -20947.397} C_VEL
LIN {X 0,Y 215.214,Z 610.234,A -85,B 0,C 180,E1 -20949.465,E2 -20949.465} C_VEL
LIN {X 0,Y 210.117,Z 612.198,A -85,B 0,C 180,E1 -20951.686,E2 -20951.686} C_VEL
LIN {X 0,Y 208.21,Z 612.988,A -85,B 0,C 180,E1 -20953.194,E2 -20953.194} C_VEL
LIN {X 0,Y 206.34,Z 614.036,A -85,B 0,C 180,E1 -20956.206,E2 -20956.206} C_VEL
LIN {X 0,Y 205.115,Z 614.174,A -85,B 0,C 180,E1 -20960.135,E2 -20960.135} C_VEL
LIN {X 0,Y 204.854,Z 612.878,A -85,B 0,C 180,E1 -20964.219,E2 -20964.219} C_VEL
LIN {X 0,Y 205.26,Z 610.289,A -85,B 0,C 180,E1 -20968.038,E2 -20968.038} C_VEL
LIN {X 0,Y 205.589,Z 608.364,A -85,B 0,C 180,E1 -20970,E2 -20970} C_VEL
LIN {X 0,Y 205.564,Z 604.428,A -85,B 0,C 180,E1 -20972.939,E2 -20972.939} C_VEL
LIN {X 0,Y 205.621,Z 599.325,A -85,B 0,C 180,E1 -20975.885,E2 -20975.885} C_VEL
LIN {X 0,Y 205.811,Z 592.894,A -85,B 0,C 180,E1 -20978.839,E2 -20978.839} C_VEL
LIN {X 0,Y 206.367,Z 584.899,A -85,B 0,C 180,E1 -20981.79,E2 -20981.79} C_VEL
LIN {X 0,Y 207.292,Z 574.973,A -85,B 0,C 180,E1 -20984.731,E2 -20984.731} C_VEL
LIN {X 0,Y 208.43,Z 564.837,A -85,B 0,C 180,E1 -20987.16,E2 -20987.16} C_VEL
LIN {X 0,Y 209.103,Z 558.949,A -85,B 0,C 180,E1 -20988.366,E2 -20988.366} C_VEL
LIN {X 0,Y 207.99,Z 548.109,A -85,B 0,C 180,E1 -20990.264,E2 -20990.264} C_VEL
LIN {X 0,Y 206.841,Z 535.122,A -85,B 0,C 180,E1 -20992.122,E2 -20992.122} C_VEL
LIN {X 0,Y 205.94,Z 521.267,A -85,B 0,C 180,E1 -20993.69,E2 -20993.69} C_VEL
LIN {X 0,Y 205.686,Z 512.508,A -85,B 0,C 180,E1 -20994.475,E2 -20994.475} C_VEL
LIN {X 0,Y 206.762,Z 507.31,A -85,B 0,C 180,E1 -20999.529,E2 -20999.529} C_VEL
LIN {X 0,Y 207.845,Z 502.786,A -85,B 0,C 180,E1 -21003.912,E2 -21003.912} C_VEL
LIN {X 0,Y 208.436,Z 500.66,A -85,B 0,C 180,E1 -21005.98,E2 -21005.98} C_VEL
LIN {X 0,Y 208.497,Z 499.257,A -85,B 0,C 180,E1 -21007.354,E2 -21007.354} C_VEL
LIN {X 0,Y 208.146,Z 496.736,A -85,B 0,C 180,E1 -21009.906,E2 -21009.906} C_VEL
LIN {X 0,Y 207.117,Z 491.43,A -85,B 0,C 180,E1 -21015.445,E2 -21015.445} C_VEL
LIN {X 0,Y 207.028,Z 490.698,A -85,B 0,C 180,E1 -21016.237,E2 -21016.237} C_VEL
LIN {X 0,Y 206.728,Z 490.731,A -85,B 0,C 180,E1 -21022.271,E2 -21022.271} C_VEL
LIN {X 0,Y 206.706,Z 490.737,A -85,B 0,C 180,E1 -21027.044,E2 -21027.044} C_VEL
LIN {X 0,Y 206.765,Z 490.724,A -85,B 0,C 180,E1 -21032.098,E2 -21032.098} C_VEL
LIN {X 0,Y 206.786,Z 490.728,A -85,B 0,C 180,E1 -21036.584,E2 -21036.584} C_VEL
LIN {X 0,Y 206.878,Z 490.713,A -85,B 0,C 180,E1 -21042.197,E2 -21042.197} C_VEL
LIN {X 0,Y 206.915,Z 490.71,A -85,B 0,C 180,E1 -21046.246,E2 -21046.246} C_VEL
LIN {X 0,Y 207.134,Z 490.68,A -85,B 0,C 180,E1 -21050.233,E2 -21050.233} C_VEL
LIN {X 0,Y 207.19,Z 490.676,A -85,B 0,C 180,E1 -21052.202,E2 -21052.202} C_VEL
LIN {X 0,Y 207.384,Z 490.648,A -85,B 0,C 180,E1 -21058.058,E2 -21058.058} C_VEL
LIN {X 0,Y 207.517,Z 490.633,A -85,B 0,C 180,E1 -21060,E2 -21060} C_VEL
LIN {X 0,Y 207.385,Z 490.651,A -85,B 0,C 180,E1 -21061.942,E2 -21061.942} C_VEL
LIN {X 0,Y 207.191,Z 490.672,A -85,B 0,C 180,E1 -21067.798,E2 -21067.798} C_VEL
LIN {X 0,Y 206.985,Z 490.701,A -85,B 0,C 180,E1 -21071.755,E2 -21071.755} C_VEL
LIN {X 0,Y 206.869,Z 490.711,A -85,B 0,C 180,E1 -21075.771,E2 -21075.771} C_VEL
LIN {X 0,Y 206.786,Z 490.726,A -85,B 0,C 180,E1 -21079.869,E2 -21079.869} C_VEL
LIN {X 0,Y 206.765,Z 490.726,A -85,B 0,C 180,E1 -21084.072,E2 -21084.072} C_VEL
LIN {X 0,Y 206.746,Z 490.733,A -85,B 0,C 180,E1 -21088.419,E2 -21088.419} C_VEL
LIN {X 0,Y 206.706,Z 490.732,A -85,B 0,C 180,E1 -21092.957,E2 -21092.957} C_VEL
LIN {X 0,Y 206.682,Z 490.739,A -85,B 0,C 180,E1 -21097.74,E2 -21097.74} C_VEL
LIN {X 0,Y 206.644,Z 490.739,A -85,B 0,C 180,E1 -21101.563,E2 -21101.563} C_VEL
LIN {X 0,Y 206.636,Z 490.744,A -85,B 0,C 180,E1 -21105.582,E2 -21105.582} C_VEL
LIN {X 0,Y 206.668,Z 490.738,A -85,B 0,C 180,E1 -21109.751,E2 -21109.751} C_VEL
LIN {X 0,Y 206.734,Z 490.733,A -85,B 0,C 180,E1 -21114.696,E2 -21114.696} C_VEL
LIN {X 0,Y 206.726,Z 490.728,A -85,B 0,C 180,E1 -21119.34,E2 -21119.34} C_VEL
LIN {X 0,Y 206.736,Z 490.733,A -85,B 0,C 180,E1 -21123.773,E2 -21123.773} C_VEL
LIN {X 0,Y 206.761,Z 490.727,A -85,B 0,C 180,E1 -21128.044,E2 -21128.044} C_VEL
LIN {X 0,Y 206.877,Z 490.717,A -85,B 0,C 180,E1 -21132.197,E2 -21132.197} C_VEL
LIN {X 0,Y 206.899,Z 490.709,A -85,B 0,C 180,E1 -21136.245,E2 -21136.245} C_VEL
LIN {X 0,Y 207.103,Z 490.688,A -85,B 0,C 180,E1 -21140.231,E2 -21140.231} C_VEL
LIN {X 0,Y 207.057,Z 490.691,A -85,B 0,C 180,E1 -21144.156,E2 -21144.156} C_VEL
LIN {X 0,Y 207.384,Z 490.653,A -85,B 0,C 180,E1 -21148.058,E2 -21148.058} C_VEL
LIN {X 0,Y 207.519,Z 490.637,A -85,B 0,C 180,E1 -21150,E2 -21150} C_VEL
LIN {X 0,Y 207.386,Z 490.652,A -85,B 0,C 180,E1 -21151.942,E2 -21151.942} C_VEL
LIN {X 0,Y 207.145,Z 490.682,A -85,B 0,C 180,E1 -21157.8,E2 -21157.8} C_VEL
LIN {X 0,Y 206.936,Z 490.708,A -85,B 0,C 180,E1 -21161.758,E2 -21161.758} C_VEL
LIN {X 0,Y 206.872,Z 490.716,A -85,B 0,C 180,E1 -21165.771,E2 -21165.771} C_VEL
LIN {X 0,Y 206.788,Z 490.726,A -85,B 0,C 180,E1 -21169.869,E2 -21169.869} C_VEL
LIN {X 0,Y 206.767,Z 490.729,A -85,B 0,C 180,E1 -21174.072,E2 -21174.072} C_VEL
LIN {X 0,Y 206.748,Z 490.729,A -85,B 0,C 180,E1 -21178.419,E2 -21178.419} C_VEL
LIN {X 0,Y 206.712,Z 490.733,A -85,B 0,C 180,E1 -21182.956,E2 -21182.956} C_VEL
LIN {X 0,Y 206.725,Z 490.734,A -85,B 0,C 180,E1 -21185.32,E2 -21185.32} C_VEL
LIN {X 0,Y 206.669,Z 490.738,A -85,B 0,C 180,E1 -21190.25,E2 -21190.25} C_VEL
LIN {X 0,Y 206.637,Z 490.744,A -85,B 0,C 180,E1 -21194.418,E2 -21194.418} C_VEL
LIN {X 0,Y 206.639,Z 490.74,A -85,B 0,C 180,E1 -21198.439,E2 -21198.439} C_VEL
LIN {X 0,Y 206.596,Z 490.75,A -85,B 0,C 180,E1 -21202.242,E2 -21202.242} C_VEL
LIN {X 0,Y 206.471,Z 490.763,A -85,B 0,C 180,E1 -21204.779,E2 -21204.779} C_VEL
LIN {X 0,Y 206.103,Z 490.81,A -85,B 0,C 180,E1 -21209.236,E2 -21209.236} C_VEL
LIN {X 0,Y 205.612,Z 490.873,A -85,B 0,C 180,E1 -21213.618,E2 -21213.618} C_VEL
LIN {X 0,Y 205.468,Z 490.894,A -85,B 0,C 180,E1 -21216.008,E2 -21216.008} C_VEL
LIN {X 0,Y 207.964,Z 506.259,A -85,B 0,C 180,E1 -21217.644,E2 -21217.644} C_VEL
LIN {X 0,Y 210.223,Z 519.27,A -85,B 0,C 180,E1 -21219.404,E2 -21219.404} C_VEL
LIN {X 0,Y 210.646,Z 522.21,A -85,B 0,C 180,E1 -21219.845,E2 -21219.845} C_VEL
LIN {X 0,Y 209.257,Z 534.316,A -85,B 0,C 180,E1 -21221.9,E2 -21221.9} C_VEL
LIN {X 0,Y 208.049,Z 544.785,A -85,B 0,C 180,E1 -21224.069,E2 -21224.069} C_VEL
LIN {X 0,Y 206.797,Z 555.263,A -85,B 0,C 180,E1 -21226.738,E2 -21226.738} C_VEL
LIN {X 0,Y 205.812,Z 564.707,A -85,B 0,C 180,E1 -21229.672,E2 -21229.672} C_VEL
LIN {X 0,Y 205.204,Z 572.52,A -85,B 0,C 180,E1 -21232.621,E2 -21232.621} C_VEL
LIN {X 0,Y 204.834,Z 579.848,A -85,B 0,C 180,E1 -21236.065,E2 -21236.065} C_VEL
LIN {X 0,Y 204.747,Z 584.827,A -85,B 0,C 180,E1 -21239.016,E2 -21239.016} C_VEL
LIN {X 0,Y 205.036,Z 589.968,A -85,B 0,C 180,E1 -21242.947,E2 -21242.947} C_VEL
LIN {X 0,Y 205.596,Z 592.742,A -85,B 0,C 180,E1 -21245.886,E2 -21245.886} C_VEL
LIN {X 0,Y 206.908,Z 595.195,A -85,B 0,C 180,E1 -21249.778,E2 -21249.778} C_VEL
LIN {X 0,Y 209.408,Z 596.227,A -85,B 0,C 180,E1 -21253.587,E2 -21253.587} C_VEL
LIN {X 0,Y 212.64,Z 595.941,A -85,B 0,C 180,E1 -21257.305,E2 -21257.305} C_VEL
LIN {X 0,Y 216.945,Z 594.327,A -85,B 0,C 180,E1 -21260.876,E2 -21260.876} C_VEL
LIN {X 0,Y 222.216,Z 591.322,A -85,B 0,C 180,E1 -21264.277,E2 -21264.277} C_VEL
LIN {X 0,Y 228.377,Z 586.96,A -85,B 0,C 180,E1 -21267.491,E2 -21267.491} C_VEL
LIN {X 0,Y 233.586,Z 582.658,A -85,B 0,C 180,E1 -21269.765,E2 -21269.765} C_VEL
LIN {X 0,Y 241.276,Z 575.576,A -85,B 0,C 180,E1 -21272.607,E2 -21272.607} C_VEL
LIN {X 0,Y 243.272,Z 573.527,A -85,B 0,C 180,E1 -21273.291,E2 -21273.291} C_VEL
LIN {X 0,Y 244.853,Z 571.635,A -85,B 0,C 180,E1 -21274.035,E2 -21274.035} C_VEL
LIN {X 0,Y 245.31,Z 570.526,A -85,B 0,C 180,E1 -21274.959,E2 -21274.959} C_VEL
LIN {X 0,Y 245.8,Z 568.601,A -85,B 0,C 180,E1 -21276.901,E2 -21276.901} C_VEL
LIN {X 0,Y 245.982,Z 567.096,A -85,B 0,C 180,E1 -21279.518,E2 -21279.518} C_VEL
LIN {X 0,Y 246.04,Z 566.579,A -85,B 0,C 180,E1 -21282.04,E2 -21282.04} C_VEL
LIN {X 0,Y 246.102,Z 566.664,A -85,B 0,C 180,E1 -21283.265,E2 -21283.265} C_VEL
LIN {X 0,Y 245.741,Z 567.844,A -85,B 0,C 180,E1 -21285.641,E2 -21285.641} C_VEL
LIN {X 0,Y 245.488,Z 568.602,A -85,B 0,C 180,E1 -21286.6,E2 -21286.6} C_VEL
LIN {X 0,Y 244.718,Z 571.01,A -85,B 0,C 180,E1 -21288.659,E2 -21288.659} C_VEL
LIN {X 0,Y 242.601,Z 575.438,A -85,B 0,C 180,E1 -21291.07,E2 -21291.07} C_VEL
LIN {X 0,Y 240.069,Z 580.404,A -85,B 0,C 180,E1 -21293.396,E2 -21293.396} C_VEL
LIN {X 0,Y 237.497,Z 584.778,A -85,B 0,C 180,E1 -21295.274,E2 -21295.274} C_VEL
LIN {X 0,Y 235.334,Z 587.824,A -85,B 0,C 180,E1 -21296.462,E2 -21296.462} C_VEL
LIN {X 0,Y 227.952,Z 595.699,A -85,B 0,C 180,E1 -21299.422,E2 -21299.422} C_VEL
LIN {X 0,Y 221.332,Z 602.072,A -85,B 0,C 180,E1 -21302.585,E2 -21302.585} C_VEL
LIN {X 0,Y 216.093,Z 606.816,A -85,B 0,C 180,E1 -21305.778,E2 -21305.778} C_VEL
LIN {X 0,Y 212.441,Z 609.904,A -85,B 0,C 180,E1 -21308.66,E2 -21308.66} C_VEL
LIN {X 0,Y 208.86,Z 612.611,A -85,B 0,C 180,E1 -21312.371,E2 -21312.371} C_VEL
LIN {X 0,Y 208.21,Z 612.988,A -85,B 0,C 180,E1 -21313.194,E2 -21313.194} C_VEL
LIN {X 0,Y 206.481,Z 613.646,A -85,B 0,C 180,E1 -21314.748,E2 -21314.748} C_VEL
LIN {X 0,Y 202.367,Z 613.939,A -85,B 0,C 180,E1 -21317.276,E2 -21317.276} C_VEL
LIN {X 0,Y 199.331,Z 613.581,A -85,B 0,C 180,E1 -21319.366,E2 -21319.366} C_VEL
LIN {X 0,Y 198.015,Z 613.074,A -85,B 0,C 180,E1 -21321.022,E2 -21321.022} C_VEL
LIN {X 0,Y 197.874,Z 612.859,A -85,B 0,C 180,E1 -21321.589,E2 -21321.589} C_VEL
LIN {X 0,Y 197.838,Z 611.807,A -85,B 0,C 180,E1 -21324.084,E2 -21324.084} C_VEL
LIN {X 0,Y 198.275,Z 608.975,A -85,B 0,C 180,E1 -21327.968,E2 -21327.968} C_VEL
LIN {X 0,Y 198.626,Z 606.885,A -85,B 0,C 180,E1 -21330,E2 -21330} C_VEL
LIN {X 0,Y 198.6,Z 602.773,A -85,B 0,C 180,E1 -21333.043,E2 -21333.043} C_VEL
LIN {X 0,Y 198.674,Z 597.381,A -85,B 0,C 180,E1 -21336.092,E2 -21336.092} C_VEL
LIN {X 0,Y 198.879,Z 590.843,A -85,B 0,C 180,E1 -21339.047,E2 -21339.047} C_VEL
LIN {X 0,Y 199.529,Z 582.273,A -85,B 0,C 180,E1 -21342.201,E2 -21342.201} C_VEL
LIN {X 0,Y 200.442,Z 571.891,A -85,B 0,C 180,E1 -21345.246,E2 -21345.246} C_VEL
LIN {X 0,Y 201.719,Z 561.414,A -85,B 0,C 180,E1 -21347.749,E2 -21347.749} C_VEL
LIN {X 0,Y 201.909,Z 557.945,A -85,B 0,C 180,E1 -21348.454,E2 -21348.454} C_VEL
LIN {X 0,Y 200.684,Z 546.525,A -85,B 0,C 180,E1 -21350.5,E2 -21350.5} C_VEL
LIN {X 0,Y 199.524,Z 532.553,A -85,B 0,C 180,E1 -21352.523,E2 -21352.523} C_VEL
LIN {X 0,Y 198.807,Z 519.431,A -85,B 0,C 180,E1 -21354.006,E2 -21354.006} C_VEL
LIN {X 0,Y 198.65,Z 512.096,A -85,B 0,C 180,E1 -21354.694,E2 -21354.694} C_VEL
LIN {X 0,Y 199.921,Z 506.239,A -85,B 0,C 180,E1 -21360.646,E2 -21360.646} C_VEL
LIN {X 0,Y 201.109,Z 501.716,A -85,B 0,C 180,E1 -21365.212,E2 -21365.212} C_VEL
LIN {X 0,Y 201.358,Z 499.305,A -85,B 0,C 180,E1 -21367.681,E2 -21367.681} C_VEL
LIN {X 0,Y 201.081,Z 497.321,A -85,B 0,C 180,E1 -21369.743,E2 -21369.743} C_VEL
LIN {X 0,Y 200.056,Z 492.138,A -85,B 0,C 180,E1 -21375.364,E2 -21375.364} C_VEL
LIN {X 0,Y 200.01,Z 491.572,A -85,B 0,C 180,E1 -21376.284,E2 -21376.284} C_VEL
LIN {X 0,Y 199.724,Z 491.606,A -85,B 0,C 180,E1 -21380.728,E2 -21380.728} C_VEL
LIN {X 0,Y 199.634,Z 491.616,A -85,B 0,C 180,E1 -21385.718,E2 -21385.718} C_VEL
LIN {X 0,Y 199.697,Z 491.609,A -85,B 0,C 180,E1 -21388.137,E2 -21388.137} C_VEL
LIN {X 0,Y 199.687,Z 491.61,A -85,B 0,C 180,E1 -21392.772,E2 -21392.772} C_VEL
LIN {X 0,Y 199.739,Z 491.603,A -85,B 0,C 180,E1 -21397.229,E2 -21397.229} C_VEL
LIN {X 0,Y 199.838,Z 491.588,A -85,B 0,C 180,E1 -21401.722,E2 -21401.722} C_VEL
LIN {X 0,Y 199.849,Z 491.589,A -85,B 0,C 180,E1 -21405.75,E2 -21405.75} C_VEL
LIN {X 0,Y 200.077,Z 491.558,A -85,B 0,C 180,E1 -21409.885,E2 -21409.885} C_VEL
LIN {X 0,Y 200.134,Z 491.553,A -85,B 0,C 180,E1 -21411.925,E2 -21411.925} C_VEL
LIN {X 0,Y 200.324,Z 491.527,A -85,B 0,C 180,E1 -21417.99,E2 -21417.99} C_VEL
LIN {X 0,Y 200.481,Z 491.51,A -85,B 0,C 180,E1 -21420,E2 -21420} C_VEL
LIN {X 0,Y 200.035,Z 491.567,A -85,B 0,C 180,E1 -21424.03,E2 -21424.03} C_VEL
LIN {X 0,Y 200.134,Z 491.552,A -85,B 0,C 180,E1 -21428.075,E2 -21428.075} C_VEL
LIN {X 0,Y 199.916,Z 491.583,A -85,B 0,C 180,E1 -21432.177,E2 -21432.177} C_VEL
LIN {X 0,Y 199.806,Z 491.593,A -85,B 0,C 180,E1 -21436.344,E2 -21436.344} C_VEL
LIN {X 0,Y 199.702,Z 491.609,A -85,B 0,C 180,E1 -21440.606,E2 -21440.606} C_VEL
LIN {X 0,Y 199.675,Z 491.609,A -85,B 0,C 180,E1 -21444.985,E2 -21444.985} C_VEL
LIN {X 0,Y 199.677,Z 491.611,A -85,B 0,C 180,E1 -21449.523,E2 -21449.523} C_VEL
LIN {X 0,Y 199.68,Z 491.609,A -85,B 0,C 180,E1 -21452.359,E2 -21452.359} C_VEL
LIN {X 0,Y 199.625,Z 491.618,A -85,B 0,C 180,E1 -21456.763,E2 -21456.763} C_VEL
LIN {X 0,Y 199.61,Z 491.618,A -85,B 0,C 180,E1 -21459.328,E2 -21459.328} C_VEL
LIN {X 0,Y 199.576,Z 491.622,A -85,B 0,C 180,E1 -21462.311,E2 -21462.311} C_VEL
LIN {X 0,Y 199.582,Z 491.622,A -85,B 0,C 180,E1 -21465.229,E2 -21465.229} C_VEL
LIN {X 0,Y 199.641,Z 491.613,A -85,B 0,C 180,E1 -21470.68,E2 -21470.68} C_VEL
LIN {X 0,Y 199.638,Z 491.617,A -85,B 0,C 180,E1 -21475.719,E2 -21475.719} C_VEL
LIN {X 0,Y 199.707,Z 491.606,A -85,B 0,C 180,E1 -21478.138,E2 -21478.138} C_VEL
LIN {X 0,Y 199.69,Z 491.61,A -85,B 0,C 180,E1 -21482.772,E2 -21482.772} C_VEL
LIN {X 0,Y 199.741,Z 491.6,A -85,B 0,C 180,E1 -21487.23,E2 -21487.23} C_VEL
LIN {X 0,Y 199.8,Z 491.597,A -85,B 0,C 180,E1 -21491.758,E2 -21491.758} C_VEL
LIN {X 0,Y 199.84,Z 491.59,A -85,B 0,C 180,E1 -21495.749,E2 -21495.749} C_VEL
LIN {X 0,Y 200.026,Z 491.569,A -85,B 0,C 180,E1 -21499.882,E2 -21499.882} C_VEL
LIN {X 0,Y 200.019,Z 491.569,A -85,B 0,C 180,E1 -21503.949,E2 -21503.949} C_VEL
LIN {X 0,Y 200.323,Z 491.532,A -85,B 0,C 180,E1 -21507.99,E2 -21507.99} C_VEL
LIN {X 0,Y 200.483,Z 491.514,A -85,B 0,C 180,E1 -21510,E2 -21510} C_VEL
LIN {X 0,Y 200.032,Z 491.565,A -85,B 0,C 180,E1 -21514.03,E2 -21514.03} C_VEL
LIN {X 0,Y 200.093,Z 491.562,A -85,B 0,C 180,E1 -21518.077,E2 -21518.077} C_VEL
LIN {X 0,Y 199.883,Z 491.583,A -85,B 0,C 180,E1 -21522.179,E2 -21522.179} C_VEL
LIN {X 0,Y 199.809,Z 491.595,A -85,B 0,C 180,E1 -21526.343,E2 -21526.343} C_VEL
LIN {X 0,Y 199.704,Z 491.605,A -85,B 0,C 180,E1 -21530.605,E2 -21530.605} C_VEL
LIN {X 0,Y 199.677,Z 491.61,A -85,B 0,C 180,E1 -21534.984,E2 -21534.984} C_VEL
LIN {X 0,Y 199.678,Z 491.611,A -85,B 0,C 180,E1 -21539.522,E2 -21539.522} C_VEL
LIN {X 0,Y 199.667,Z 491.611,A -85,B 0,C 180,E1 -21542.352,E2 -21542.352} C_VEL
LIN {X 0,Y 199.643,Z 491.614,A -85,B 0,C 180,E1 -21546.759,E2 -21546.759} C_VEL
LIN {X 0,Y 199.642,Z 491.613,A -85,B 0,C 180,E1 -21549.321,E2 -21549.321} C_VEL
LIN {X 0,Y 199.583,Z 491.622,A -85,B 0,C 180,E1 -21554.771,E2 -21554.771} C_VEL
LIN {X 0,Y 199.577,Z 491.621,A -85,B 0,C 180,E1 -21558.004,E2 -21558.004} C_VEL
LIN {X 0,Y 199.584,Z 491.621,A -85,B 0,C 180,E1 -21560.778,E2 -21560.778} C_VEL
LIN {X 0,Y 199.333,Z 491.654,A -85,B 0,C 180,E1 -21565.658,E2 -21565.658} C_VEL
LIN {X 0,Y 199.167,Z 491.674,A -85,B 0,C 180,E1 -21568.041,E2 -21568.041} C_VEL
LIN {X 0,Y 198.688,Z 491.738,A -85,B 0,C 180,E1 -21572.623,E2 -21572.623} C_VEL
LIN {X 0,Y 198.434,Z 491.844,A -85,B 0,C 180,E1 -21575.899,E2 -21575.899} C_VEL
LIN {X 0,Y 200.758,Z 506.272,A -85,B 0,C 180,E1 -21577.474,E2 -21577.474} C_VEL
LIN {X 0,Y 202.963,Z 518.906,A -85,B 0,C 180,E1 -21579.218,E2 -21579.218} C_VEL
LIN {X 0,Y 203.513,Z 522.636,A -85,B 0,C 180,E1 -21579.797,E2 -21579.797} C_VEL
LIN {X 0,Y 202.073,Z 535.082,A -85,B 0,C 180,E1 -21582.021,E2 -21582.021} C_VEL
LIN {X 0,Y 200.819,Z 545.379,A -85,B 0,C 180,E1 -21584.262,E2 -21584.262} C_VEL
LIN {X 0,Y 199.551,Z 556.7,A -85,B 0,C 180,E1 -21587.284,E2 -21587.284} C_VEL
LIN {X 0,Y 198.569,Z 565.986,A -85,B 0,C 180,E1 -21590.321,E2 -21590.321} C_VEL
LIN {X 0,Y 198.103,Z 572.659,A -85,B 0,C 180,E1 -21592.969,E2 -21592.969} C_VEL
LIN {X 0,Y 197.788,Z 578.862,A -85,B 0,C 180,E1 -21595.924,E2 -21595.924} C_VEL
LIN {X 0,Y 197.683,Z 584.133,A -85,B 0,C 180,E1 -21598.981,E2 -21598.981} C_VEL
LIN {X 0,Y 197.854,Z 588.376,A -85,B 0,C 180,E1 -21602.035,E2 -21602.035} C_VEL
LIN {X 0,Y 198.164,Z 590.674,A -85,B 0,C 180,E1 -21604.067,E2 -21604.067} C_VEL
LIN {X 0,Y 199.09,Z 594.117,A -85,B 0,C 180,E1 -21608.117,E2 -21608.117} C_VEL
LIN {X 0,Y 201.112,Z 596.194,A -85,B 0,C 180,E1 -21612.103,E2 -21612.103} C_VEL
LIN {X 0,Y 204.078,Z 596.933,A -85,B 0,C 180,E1 -21615.992,E2 -21615.992} C_VEL
LIN {X 0,Y 208.063,Z 596.314,A -85,B 0,C 180,E1 -21619.742,E2 -21619.742} C_VEL
LIN {X 0,Y 213.063,Z 594.38,A -85,B 0,C 180,E1 -21623.317,E2 -21623.317} C_VEL
LIN {X 0,Y 218.992,Z 591.186,A -85,B 0,C 180,E1 -21626.698,E2 -21626.698} C_VEL
LIN {X 0,Y 225.88,Z 586.538,A -85,B 0,C 180,E1 -21629.856,E2 -21629.856} C_VEL
LIN {X 0,Y 233.678,Z 580.351,A -85,B 0,C 180,E1 -21632.776,E2 -21632.776} C_VEL
LIN {X 0,Y 238.637,Z 575.93,A -85,B 0,C 180,E1 -21634.45,E2 -21634.45} C_VEL
LIN {X 0,Y 239.856,Z 574.088,A -85,B 0,C 180,E1 -21635.875,E2 -21635.875} C_VEL
LIN {X 0,Y 240.395,Z 572.587,A -85,B 0,C 180,E1 -21637.875,E2 -21637.875} C_VEL
LIN {X 0,Y 240.703,Z 571.516,A -85,B 0,C 180,E1 -21640.611,E2 -21640.611} C_VEL
LIN {X 0,Y 240.839,Z 571.431,A -85,B 0,C 180,E1 -21643.152,E2 -21643.152} C_VEL
LIN {X 0,Y 240.449,Z 572.527,A -85,B 0,C 180,E1 -21645.453,E2 -21645.453} C_VEL
LIN {X 0,Y 239.374,Z 575.214,A -85,B 0,C 180,E1 -21648.168,E2 -21648.168} C_VEL
LIN {X 0,Y 237.155,Z 578.999,A -85,B 0,C 180,E1 -21650.399,E2 -21650.399} C_VEL
LIN {X 0,Y 233.874,Z 584.291,A -85,B 0,C 180,E1 -21653.058,E2 -21653.058} C_VEL
LIN {X 0,Y 231.252,Z 587.953,A -85,B 0,C 180,E1 -21654.73,E2 -21654.73} C_VEL
LIN {X 0,Y 229.643,Z 589.794,A -85,B 0,C 180,E1 -21655.516,E2 -21655.516} C_VEL
LIN {X 0,Y 221.986,Z 597.138,A -85,B 0,C 180,E1 -21658.507,E2 -21658.507} C_VEL
LIN {X 0,Y 215.12,Z 603.032,A -85,B 0,C 180,E1 -21661.724,E2 -21661.724} C_VEL
LIN {X 0,Y 210.686,Z 606.545,A -85,B 0,C 180,E1 -21664.3,E2 -21664.3} C_VEL
LIN {X 0,Y 205.852,Z 610.14,A -85,B 0,C 180,E1 -21667.941,E2 -21667.941} C_VEL
LIN {X 0,Y 202.107,Z 612.46,A -85,B 0,C 180,E1 -21671.762,E2 -21671.762} C_VEL
LIN {X 0,Y 199.429,Z 613.537,A -85,B 0,C 180,E1 -21675.718,E2 -21675.718} C_VEL
LIN {X 0,Y 198.135,Z 613.362,A -85,B 0,C 180,E1 -21679.784,E2 -21679.784} C_VEL
LIN {X 0,Y 197.874,Z 612.859,A -85,B 0,C 180,E1 -21681.589,E2 -21681.589} C_VEL
LIN {X 0,Y 197.199,Z 612.119,A -85,B 0,C 180,E1 -21683.275,E2 -21683.275} C_VEL
LIN {X 0,Y 195.812,Z 610.933,A -85,B 0,C 180,E1 -21684.921,E2 -21684.921} C_VEL
LIN {X 0,Y 192.654,Z 607.572,A -85,B 0,C 180,E1 -21688.184,E2 -21688.184} C_VEL
LIN {X 0,Y 191.685,Z 604.825,A -85,B 0,C 180,E1 -21690.401,E2 -21690.401} C_VEL
LIN {X 0,Y 191.668,Z 600.945,A -85,B 0,C 180,E1 -21693.153,E2 -21693.153} C_VEL
LIN {X 0,Y 191.735,Z 595.333,A -85,B 0,C 180,E1 -21696.313,E2 -21696.313} C_VEL
LIN {X 0,Y 191.951,Z 588.52,A -85,B 0,C 180,E1 -21699.377,E2 -21699.377} C_VEL
LIN {X 0,Y 192.677,Z 579.469,A -85,B 0,C 180,E1 -21702.641,E2 -21702.641} C_VEL
LIN {X 0,Y 193.474,Z 570.57,A -85,B 0,C 180,E1 -21705.269,E2 -21705.269} C_VEL
LIN {X 0,Y 194.763,Z 559.917,A -85,B 0,C 180,E1 -21707.862,E2 -21707.862} C_VEL
LIN {X 0,Y 194.63,Z 555.929,A -85,B 0,C 180,E1 -21708.691,E2 -21708.691} C_VEL
LIN {X 0,Y 193.204,Z 542.293,A -85,B 0,C 180,E1 -21711.113,E2 -21711.113} C_VEL
LIN {X 0,Y 192.176,Z 528.905,A -85,B 0,C 180,E1 -21713.007,E2 -21713.007} C_VEL
LIN {X 0,Y 191.581,Z 515.218,A -85,B 0,C 180,E1 -21714.519,E2 -21714.519} C_VEL
LIN {X 0,Y 191.573,Z 511.732,A -85,B 0,C 180,E1 -21714.881,E2 -21714.881} C_VEL
LIN {X 0,Y 192.813,Z 506.26,A -85,B 0,C 180,E1 -21720.684,E2 -21720.684} C_VEL
LIN {X 0,Y 194.048,Z 501.772,A -85,B 0,C 180,E1 -21725.414,E2 -21725.414} C_VEL
LIN {X 0,Y 194.25,Z 499.386,A -85,B 0,C 180,E1 -21727.956,E2 -21727.956} C_VEL
LIN {X 0,Y 193.527,Z 495.647,A -85,B 0,C 180,E1 -21732.07,E2 -21732.07} C_VEL
LIN {X 0,Y 192.966,Z 492.45,A -85,B 0,C 180,E1 -21735.849,E2 -21735.849} C_VEL
LIN {X 0,Y 192.625,Z 492.486,A -85,B 0,C 180,E1 -21741.666,E2 -21741.666} C_VEL
LIN {X 0,Y 192.598,Z 492.495,A -85,B 0,C 180,E1 -21746.814,E2 -21746.814} C_VEL
LIN {X 0,Y 192.661,Z 492.48,A -85,B 0,C 180,E1 -21751.692,E2 -21751.692} C_VEL
LIN {X 0,Y 192.707,Z 492.481,A -85,B 0,C 180,E1 -21756.349,E2 -21756.349} C_VEL
LIN {X 0,Y 192.782,Z 492.467,A -85,B 0,C 180,E1 -21761.414,E2 -21761.414} C_VEL
LIN {X 0,Y 192.855,Z 492.458,A -85,B 0,C 180,E1 -21767.37,E2 -21767.37} C_VEL
LIN {X 0,Y 193.081,Z 492.432,A -85,B 0,C 180,E1 -21771.628,E2 -21771.628} C_VEL
LIN {X 0,Y 193.266,Z 492.406,A -85,B 0,C 180,E1 -21777.916,E2 -21777.916} C_VEL
LIN {X 0,Y 193.445,Z 492.386,A -85,B 0,C 180,E1 -21780,E2 -21780} C_VEL
LIN {X 0,Y 192.982,Z 492.446,A -85,B 0,C 180,E1 -21784.177,E2 -21784.177} C_VEL
LIN {X 0,Y 193.081,Z 492.432,A -85,B 0,C 180,E1 -21788.372,E2 -21788.372} C_VEL
LIN {X 0,Y 192.855,Z 492.461,A -85,B 0,C 180,E1 -21792.63,E2 -21792.63} C_VEL
LIN {X 0,Y 192.759,Z 492.472,A -85,B 0,C 180,E1 -21796.959,E2 -21796.959} C_VEL
LIN {X 0,Y 192.638,Z 492.487,A -85,B 0,C 180,E1 -21801.398,E2 -21801.398} C_VEL
LIN {X 0,Y 192.666,Z 492.482,A -85,B 0,C 180,E1 -21804.225,E2 -21804.225} C_VEL
LIN {X 0,Y 192.652,Z 492.486,A -85,B 0,C 180,E1 -21808.893,E2 -21808.893} C_VEL
LIN {X 0,Y 192.601,Z 492.488,A -85,B 0,C 180,E1 -21813.186,E2 -21813.186} C_VEL
LIN {X 0,Y 192.553,Z 492.5,A -85,B 0,C 180,E1 -21818.352,E2 -21818.352} C_VEL
LIN {X 0,Y 192.493,Z 492.504,A -85,B 0,C 180,E1 -21823.096,E2 -21823.096} C_VEL
LIN {X 0,Y 192.495,Z 492.505,A -85,B 0,C 180,E1 -21826.904,E2 -21826.904} C_VEL
LIN {X 0,Y 192.576,Z 492.492,A -85,B 0,C 180,E1 -21831.654,E2 -21831.654} C_VEL
LIN {X 0,Y 192.601,Z 492.495,A -85,B 0,C 180,E1 -21834.279,E2 -21834.279} C_VEL
LIN {X 0,Y 192.61,Z 492.486,A -85,B 0,C 180,E1 -21839.281,E2 -21839.281} C_VEL
LIN {X 0,Y 192.667,Z 492.483,A -85,B 0,C 180,E1 -21841.693,E2 -21841.693} C_VEL
LIN {X 0,Y 192.709,Z 492.478,A -85,B 0,C 180,E1 -21846.349,E2 -21846.349} C_VEL
LIN {X 0,Y 192.735,Z 492.475,A -85,B 0,C 180,E1 -21851.458,E2 -21851.458} C_VEL
LIN {X 0,Y 192.768,Z 492.47,A -85,B 0,C 180,E1 -21855.214,E2 -21855.214} C_VEL
LIN {X 0,Y 192.948,Z 492.449,A -85,B 0,C 180,E1 -21859.567,E2 -21859.567} C_VEL
LIN {X 0,Y 192.982,Z 492.446,A -85,B 0,C 180,E1 -21863.728,E2 -21863.728} C_VEL
LIN {X 0,Y 193.265,Z 492.41,A -85,B 0,C 180,E1 -21867.916,E2 -21867.916} C_VEL
LIN {X 0,Y 193.447,Z 492.39,A -85,B 0,C 180,E1 -21870,E2 -21870} C_VEL
LIN {X 0,Y 192.978,Z 492.443,A -85,B 0,C 180,E1 -21874.177,E2 -21874.177} C_VEL
LIN {X 0,Y 193.04,Z 492.439,A -85,B 0,C 180,E1 -21878.374,E2 -21878.374} C_VEL
LIN {X 0,Y 192.809,Z 492.462,A -85,B 0,C 180,E1 -21882.633,E2 -21882.633} C_VEL
LIN {X 0,Y 192.762,Z 492.472,A -85,B 0,C 180,E1 -21886.959,E2 -21886.959} C_VEL
LIN {X 0,Y 192.641,Z 492.485,A -85,B 0,C 180,E1 -21891.397,E2 -21891.397} C_VEL
LIN {X 0,Y 192.668,Z 492.485,A -85,B 0,C 180,E1 -21894.225,E2 -21894.225} C_VEL
LIN {X 0,Y 192.653,Z 492.484,A -85,B 0,C 180,E1 -21898.892,E2 -21898.892} C_VEL
LIN {X 0,Y 192.604,Z 492.491,A -85,B 0,C 180,E1 -21903.185,E2 -21903.185} C_VEL
LIN {X 0,Y 192.613,Z 492.49,A -85,B 0,C 180,E1 -21906.607,E2 -21906.607} C_VEL
LIN {X 0,Y 192.527,Z 492.499,A -85,B 0,C 180,E1 -21911.077,E2 -21911.077} C_VEL
LIN {X 0,Y 192.493,Z 492.505,A -85,B 0,C 180,E1 -21916.076,E2 -21916.076} C_VEL
LIN {X 0,Y 192.499,Z 492.505,A -85,B 0,C 180,E1 -21920.059,E2 -21920.059} C_VEL
LIN {X 0,Y 192.386,Z 492.519,A -85,B 0,C 180,E1 -21924.232,E2 -21924.232} C_VEL
LIN {X 0,Y 192.16,Z 492.544,A -85,B 0,C 180,E1 -21927.267,E2 -21927.267} C_VEL
LIN {X 0,Y 191.708,Z 492.607,A -85,B 0,C 180,E1 -21931.624,E2 -21931.624} C_VEL
LIN {X 0,Y 191.394,Z 492.645,A -85,B 0,C 180,E1 -21935.765,E2 -21935.765} C_VEL
LIN {X 0,Y 193.755,Z 507.384,A -85,B 0,C 180,E1 -21937.472,E2 -21937.472} C_VEL
LIN {X 0,Y 196.086,Z 520.608,A -85,B 0,C 180,E1 -21939.403,E2 -21939.403} C_VEL
LIN {X 0,Y 196.153,Z 524.824,A -85,B 0,C 180,E1 -21940.1,E2 -21940.1} C_VEL
LIN {X 0,Y 194.695,Z 536.963,A -85,B 0,C 180,E1 -21942.403,E2 -21942.403} C_VEL
LIN {X 0,Y 193.47,Z 547.01,A -85,B 0,C 180,E1 -21944.73,E2 -21944.73} C_VEL
LIN {X 0,Y 192.472,Z 556.387,A -85,B 0,C 180,E1 -21947.344,E2 -21947.344} C_VEL
LIN {X 0,Y 191.493,Z 565.671,A -85,B 0,C 180,E1 -21950.493,E2 -21950.493} C_VEL
LIN {X 0,Y 190.925,Z 573.388,A -85,B 0,C 180,E1 -21953.659,E2 -21953.659} C_VEL
LIN {X 0,Y 190.711,Z 579.75,A -85,B 0,C 180,E1 -21956.831,E2 -21956.831} C_VEL
LIN {X 0,Y 190.631,Z 584.909,A -85,B 0,C 180,E1 -21960,E2 -21960} C_VEL
LIN {X 0,Y 191.115,Z 590.219,A -85,B 0,C 180,E1 -21964.217,E2 -21964.217} C_VEL
LIN {X 0,Y 192.074,Z 594.03,A -85,B 0,C 180,E1 -21968.416,E2 -21968.416} C_VEL
LIN {X 0,Y 194.194,Z 596.428,A -85,B 0,C 180,E1 -21972.541,E2 -21972.541} C_VEL
LIN {X 0,Y 197.285,Z 597.485,A -85,B 0,C 180,E1 -21976.558,E2 -21976.558} C_VEL
LIN {X 0,Y 201.475,Z 597.246,A -85,B 0,C 180,E1 -21980.415,E2 -21980.415} C_VEL
LIN {X 0,Y 206.697,Z 595.749,A -85,B 0,C 180,E1 -21984.08,E2 -21984.08} C_VEL
LIN {X 0,Y 212.864,Z 592.927,A -85,B 0,C 180,E1 -21987.531,E2 -21987.531} C_VEL
LIN {X 0,Y 220.006,Z 588.778,A -85,B 0,C 180,E1 -21990.738,E2 -21990.738} C_VEL
LIN {X 0,Y 228.11,Z 583.179,A -85,B 0,C 180,E1 -21993.681,E2 -21993.681} C_VEL
LIN {X 0,Y 232.365,Z 579.803,A -85,B 0,C 180,E1 -21995.076,E2 -21995.076} C_VEL
LIN {X 0,Y 233.504,Z 578.725,A -85,B 0,C 180,E1 -21995.644,E2 -21995.644} C_VEL
LIN {X 0,Y 234.333,Z 577.626,A -85,B 0,C 180,E1 -21996.858,E2 -21996.858} C_VEL
LIN {X 0,Y 234.862,Z 576.481,A -85,B 0,C 180,E1 -21998.932,E2 -21998.932} C_VEL
LIN {X 0,Y 235.236,Z 575.89,A -85,B 0,C 180,E1 -22001.676,E2 -22001.676} C_VEL
LIN {X 0,Y 235.206,Z 576.316,A -85,B 0,C 180,E1 -22004.182,E2 -22004.182} C_VEL
LIN {X 0,Y 234.448,Z 577.923,A -85,B 0,C 180,E1 -22006.412,E2 -22006.412} C_VEL
LIN {X 0,Y 233.973,Z 578.964,A -85,B 0,C 180,E1 -22007.48,E2 -22007.48} C_VEL
LIN {X 0,Y 232.201,Z 581.495,A -85,B 0,C 180,E1 -22009.172,E2 -22009.172} C_VEL
LIN {X 0,Y 229.724,Z 584.974,A -85,B 0,C 180,E1 -22011.159,E2 -22011.159} C_VEL
LIN {X 0,Y 227.184,Z 588.255,A -85,B 0,C 180,E1 -22012.898,E2 -22012.898} C_VEL
LIN {X 0,Y 224.01,Z 591.747,A -85,B 0,C 180,E1 -22014.52,E2 -22014.52} C_VEL
LIN {X 0,Y 216.055,Z 598.475,A -85,B 0,C 180,E1 -22017.539,E2 -22017.539} C_VEL
LIN {X 0,Y 208.959,Z 603.872,A -85,B 0,C 180,E1 -22020.811,E2 -22020.811} C_VEL
LIN {X 0,Y 204.332,Z 607.063,A -85,B 0,C 180,E1 -22023.44,E2 -22023.44} C_VEL
LIN {X 0,Y 199.301,Z 610.241,A -85,B 0,C 180,E1 -22027.176,E2 -22027.176} C_VEL
LIN {X 0,Y 195.38,Z 612.23,A -85,B 0,C 180,E1 -22031.11,E2 -22031.11} C_VEL
LIN {X 0,Y 192.541,Z 612.988,A -85,B 0,C 180,E1 -22035.196,E2 -22035.196} C_VEL
LIN {X 0,Y 191.17,Z 612.52,A -85,B 0,C 180,E1 -22039.408,E2 -22039.408} C_VEL
LIN {X 0,Y 190.848,Z 610.606,A -85,B 0,C 180,E1 -22043.868,E2 -22043.868} C_VEL
LIN {X 0,Y 191.313,Z 607.559,A -85,B 0,C 180,E1 -22047.894,E2 -22047.894} C_VEL
LIN {X 0,Y 191.685,Z 604.825,A -85,B 0,C 180,E1 -22050.401,E2 -22050.401} C_VEL
LIN {X 0,Y 191.003,Z 602.525,A -85,B 0,C 180,E1 -22052.003,E2 -22052.003} C_VEL
LIN {X 0,Y 189.454,Z 599.808,A -85,B 0,C 180,E1 -22053.524,E2 -22053.524} C_VEL
LIN {X 0,Y 185.481,Z 592.407,A -85,B 0,C 180,E1 -22056.962,E2 -22056.962} C_VEL
LIN {X 0,Y 184.94,Z 588.92,A -85,B 0,C 180,E1 -22058.478,E2 -22058.478} C_VEL
LIN {X 0,Y 185.574,Z 579.815,A -85,B 0,C 180,E1 -22062.022,E2 -22062.022} C_VEL
LIN {X 0,Y 186.317,Z 571.158,A -85,B 0,C 180,E1 -22064.751,E2 -22064.751} C_VEL
LIN {X 0,Y 187.491,Z 560.741,A -85,B 0,C 180,E1 -22067.45,E2 -22067.45} C_VEL
LIN {X 0,Y 187.802,Z 558.377,A -85,B 0,C 180,E1 -22067.983,E2 -22067.983} C_VEL
LIN {X 0,Y 186.474,Z 546.066,A -85,B 0,C 180,E1 -22070.402,E2 -22070.402} C_VEL
LIN {X 0,Y 185.3,Z 532.518,A -85,B 0,C 180,E1 -22072.544,E2 -22072.544} C_VEL
LIN {X 0,Y 184.643,Z 519.564,A -85,B 0,C 180,E1 -22074.169,E2 -22074.169} C_VEL
LIN {X 0,Y 184.486,Z 511.377,A -85,B 0,C 180,E1 -22075,E2 -22075} C_VEL
LIN {X 0,Y 185.724,Z 506.231,A -85,B 0,C 180,E1 -22080.721,E2 -22080.721} C_VEL
LIN {X 0,Y 186.965,Z 501.771,A -85,B 0,C 180,E1 -22085.637,E2 -22085.637} C_VEL
LIN {X 0,Y 187.164,Z 499.697,A -85,B 0,C 180,E1 -22087.95,E2 -22087.95} C_VEL
LIN {X 0,Y 186.311,Z 495.502,A -85,B 0,C 180,E1 -22092.765,E2 -22092.765} C_VEL
LIN {X 0,Y 185.944,Z 493.324,A -85,B 0,C 180,E1 -22095.6,E2 -22095.6} C_VEL
LIN {X 0,Y 185.636,Z 493.359,A -85,B 0,C 180,E1 -22099.939,E2 -22099.939} C_VEL
LIN {X 0,Y 185.576,Z 493.365,A -85,B 0,C 180,E1 -22102.704,E2 -22102.704} C_VEL
LIN {X 0,Y 185.541,Z 493.372,A -85,B 0,C 180,E1 -22107.975,E2 -22107.975} C_VEL
LIN {X 0,Y 185.581,Z 493.365,A -85,B 0,C 180,E1 -22110.577,E2 -22110.577} C_VEL
LIN {X 0,Y 185.588,Z 493.366,A -85,B 0,C 180,E1 -22115.383,E2 -22115.383} C_VEL
LIN {X 0,Y 185.695,Z 493.351,A -85,B 0,C 180,E1 -22121.116,E2 -22121.116} C_VEL
LIN {X 0,Y 185.729,Z 493.351,A -85,B 0,C 180,E1 -22124.64,E2 -22124.64} C_VEL
LIN {X 0,Y 185.944,Z 493.318,A -85,B 0,C 180,E1 -22129.329,E2 -22129.329} C_VEL
LIN {X 0,Y 185.97,Z 493.318,A -85,B 0,C 180,E1 -22133.491,E2 -22133.491} C_VEL
LIN {X 0,Y 186.21,Z 493.284,A -85,B 0,C 180,E1 -22137.837,E2 -22137.837} C_VEL
LIN {X 0,Y 186.409,Z 493.262,A -85,B 0,C 180,E1 -22140,E2 -22140} C_VEL
LIN {X 0,Y 185.93,Z 493.325,A -85,B 0,C 180,E1 -22144.336,E2 -22144.336} C_VEL
LIN {X 0,Y 186.031,Z 493.312,A -85,B 0,C 180,E1 -22148.692,E2 -22148.692} C_VEL
LIN {X 0,Y 185.767,Z 493.342,A -85,B 0,C 180,E1 -22153.121,E2 -22153.121} C_VEL
LIN {X 0,Y 185.676,Z 493.356,A -85,B 0,C 180,E1 -22158.868,E2 -22158.868} C_VEL
LIN {X 0,Y 185.602,Z 493.363,A -85,B 0,C 180,E1 -22164.663,E2 -22164.663} C_VEL
LIN {X 0,Y 185.581,Z 493.367,A -85,B 0,C 180,E1 -22169.493,E2 -22169.493} C_VEL
LIN {X 0,Y 185.502,Z 493.377,A -85,B 0,C 180,E1 -22174.632,E2 -22174.632} C_VEL
LIN {X 0,Y 185.507,Z 493.376,A -85,B 0,C 180,E1 -22177.313,E2 -22177.313} C_VEL
LIN {X 0,Y 185.473,Z 493.377,A -85,B 0,C 180,E1 -22180.725,E2 -22180.725} C_VEL
LIN {X 0,Y 185.481,Z 493.381,A -85,B 0,C 180,E1 -22186.049,E2 -22186.049} C_VEL
LIN {X 0,Y 185.492,Z 493.377,A -85,B 0,C 180,E1 -22189.902,E2 -22189.902} C_VEL
LIN {X 0,Y 185.546,Z 493.371,A -85,B 0,C 180,E1 -22192.697,E2 -22192.697} C_VEL
LIN {X 0,Y 185.548,Z 493.371,A -85,B 0,C 180,E1 -22197.976,E2 -22197.976} C_VEL
LIN {X 0,Y 185.585,Z 493.366,A -85,B 0,C 180,E1 -22200.576,E2 -22200.576} C_VEL
LIN {X 0,Y 185.591,Z 493.365,A -85,B 0,C 180,E1 -22205.383,E2 -22205.383} C_VEL
LIN {X 0,Y 185.61,Z 493.363,A -85,B 0,C 180,E1 -22210.076,E2 -22210.076} C_VEL
LIN {X 0,Y 185.699,Z 493.351,A -85,B 0,C 180,E1 -22214.638,E2 -22214.638} C_VEL
LIN {X 0,Y 185.891,Z 493.327,A -85,B 0,C 180,E1 -22219.419,E2 -22219.419} C_VEL
LIN {X 0,Y 185.945,Z 493.321,A -85,B 0,C 180,E1 -22223.49,E2 -22223.49} C_VEL
LIN {X 0,Y 186.209,Z 493.288,A -85,B 0,C 180,E1 -22227.837,E2 -22227.837} C_VEL
LIN {X 0,Y 186.411,Z 493.267,A -85,B 0,C 180,E1 -22230,E2 -22230} C_VEL
LIN {X 0,Y 185.924,Z 493.321,A -85,B 0,C 180,E1 -22234.336,E2 -22234.336} C_VEL
LIN {X 0,Y 185.987,Z 493.316,A -85,B 0,C 180,E1 -22238.694,E2 -22238.694} C_VEL
LIN {X 0,Y 185.735,Z 493.343,A -85,B 0,C 180,E1 -22243.123,E2 -22243.123} C_VEL
LIN {X 0,Y 185.694,Z 493.354,A -85,B 0,C 180,E1 -22247.625,E2 -22247.625} C_VEL
LIN {X 0,Y 185.601,Z 493.362,A -85,B 0,C 180,E1 -22252.251,E2 -22252.251} C_VEL
LIN {X 0,Y 185.566,Z 493.369,A -85,B 0,C 180,E1 -22257.032,E2 -22257.032} C_VEL
LIN {X 0,Y 185.582,Z 493.366,A -85,B 0,C 180,E1 -22259.493,E2 -22259.493} C_VEL
LIN {X 0,Y 185.523,Z 493.374,A -85,B 0,C 180,E1 -22264.628,E2 -22264.628} C_VEL
LIN {X 0,Y 185.547,Z 493.371,A -85,B 0,C 180,E1 -22267.304,E2 -22267.304} C_VEL
LIN {X 0,Y 185.488,Z 493.376,A -85,B 0,C 180,E1 -22270.73,E2 -22270.73} C_VEL
LIN {X 0,Y 185.482,Z 493.381,A -85,B 0,C 180,E1 -22273.951,E2 -22273.951} C_VEL
LIN {X 0,Y 185.46,Z 493.379,A -85,B 0,C 180,E1 -22279.28,E2 -22279.28} C_VEL
LIN {X 0,Y 185.367,Z 493.393,A -85,B 0,C 180,E1 -22282.769,E2 -22282.769} C_VEL
LIN {X 0,Y 185.148,Z 493.416,A -85,B 0,C 180,E1 -22286.626,E2 -22286.626} C_VEL
LIN {X 0,Y 184.692,Z 493.478,A -85,B 0,C 180,E1 -22291.071,E2 -22291.071} C_VEL
LIN {X 0,Y 184.369,Z 493.648,A -85,B 0,C 180,E1 -22295.68,E2 -22295.68} C_VEL
LIN {X 0,Y 186.675,Z 507.95,A -85,B 0,C 180,E1 -22297.399,E2 -22297.399} C_VEL
LIN {X 0,Y 189.124,Z 521.916,A -85,B 0,C 180,E1 -22299.537,E2 -22299.537} C_VEL
LIN {X 0,Y 188.519,Z 529.857,A -85,B 0,C 180,E1 -22300.961,E2 -22300.961} C_VEL
LIN {X 0,Y 186.972,Z 542.149,A -85,B 0,C 180,E1 -22303.625,E2 -22303.625} C_VEL
LIN {X 0,Y 185.741,Z 552.26,A -85,B 0,C 180,E1 -22306.32,E2 -22306.32} C_VEL
LIN {X 0,Y 184.841,Z 560.809,A -85,B 0,C 180,E1 -22309.04,E2 -22309.04} C_VEL
LIN {X 0,Y 184.137,Z 569.429,A -85,B 0,C 180,E1 -22312.323,E2 -22312.323} C_VEL
LIN {X 0,Y 183.703,Z 576.512,A -85,B 0,C 180,E1 -22315.611,E2 -22315.611} C_VEL
LIN {X 0,Y 183.589,Z 582.315,A -85,B 0,C 180,E1 -22318.903,E2 -22318.903} C_VEL
LIN {X 0,Y 183.734,Z 587.061,A -85,B 0,C 180,E1 -22322.192,E2 -22322.192} C_VEL
LIN {X 0,Y 184.24,Z 590.858,A -85,B 0,C 180,E1 -22325.472,E2 -22325.472} C_VEL
LIN {X 0,Y 185.583,Z 594.803,A -85,B 0,C 180,E1 -22330.06,E2 -22330.06} C_VEL
LIN {X 0,Y 187.29,Z 596.538,A -85,B 0,C 180,E1 -22333.011,E2 -22333.011} C_VEL
LIN {X 0,Y 190.526,Z 597.971,A -85,B 0,C 180,E1 -22337.163,E2 -22337.163} C_VEL
LIN {X 0,Y 194.914,Z 598.12,A -85,B 0,C 180,E1 -22341.135,E2 -22341.135} C_VEL
LIN {X 0,Y 200.336,Z 596.979,A -85,B 0,C 180,E1 -22344.896,E2 -22344.896} C_VEL
LIN {X 0,Y 206.773,Z 594.609,A -85,B 0,C 180,E1 -22348.414,E2 -22348.414} C_VEL
LIN {X 0,Y 214.194,Z 590.932,A -85,B 0,C 180,E1 -22351.667,E2 -22351.667} C_VEL
LIN {X 0,Y 222.553,Z 585.846,A -85,B 0,C 180,E1 -22354.64,E2 -22354.64} C_VEL
LIN {X 0,Y 226.957,Z 582.78,A -85,B 0,C 180,E1 -22356.04,E2 -22356.04} C_VEL
LIN {X 0,Y 228.18,Z 581.783,A -85,B 0,C 180,E1 -22356.792,E2 -22356.792} C_VEL
LIN {X 0,Y 228.692,Z 581.103,A -85,B 0,C 180,E1 -22357.925,E2 -22357.925} C_VEL
LIN {X 0,Y 229.245,Z 580.371,A -85,B 0,C 180,E1 -22360.076,E2 -22360.076} C_VEL
LIN {X 0,Y 229.589,Z 580.263,A -85,B 0,C 180,E1 -22362.72,E2 -22362.72} C_VEL
LIN {X 0,Y 229.124,Z 581.275,A -85,B 0,C 180,E1 -22365.131,E2 -22365.131} C_VEL
LIN {X 0,Y 227.958,Z 583.122,A -85,B 0,C 180,E1 -22367.291,E2 -22367.291} C_VEL
LIN {X 0,Y 224.443,Z 587.317,A -85,B 0,C 180,E1 -22370.065,E2 -22370.065} C_VEL
LIN {X 0,Y 221.767,Z 590.373,A -85,B 0,C 180,E1 -22371.831,E2 -22371.831} C_VEL
LIN {X 0,Y 220.256,Z 591.901,A -85,B 0,C 180,E1 -22372.68,E2 -22372.68} C_VEL
LIN {X 0,Y 216.361,Z 595.2,A -85,B 0,C 180,E1 -22374.219,E2 -22374.219} C_VEL
LIN {X 0,Y 208.26,Z 601.08,A -85,B 0,C 180,E1 -22377.32,E2 -22377.32} C_VEL
LIN {X 0,Y 201.189,Z 605.675,A -85,B 0,C 180,E1 -22380.721,E2 -22380.721} C_VEL
LIN {X 0,Y 195.233,Z 609.036,A -85,B 0,C 180,E1 -22384.407,E2 -22384.407} C_VEL
LIN {X 0,Y 190.553,Z 611.227,A -85,B 0,C 180,E1 -22388.357,E2 -22388.357} C_VEL
LIN {X 0,Y 187.022,Z 612.247,A -85,B 0,C 180,E1 -22392.504,E2 -22392.504} C_VEL
LIN {X 0,Y 184.85,Z 612.075,A -85,B 0,C 180,E1 -22396.813,E2 -22396.813} C_VEL
LIN {X 0,Y 183.898,Z 610.687,A -85,B 0,C 180,E1 -22401.207,E2 -22401.207} C_VEL
LIN {X 0,Y 183.995,Z 607.958,A -85,B 0,C 180,E1 -22405.618,E2 -22405.618} C_VEL
LIN {X 0,Y 184.588,Z 604.922,A -85,B 0,C 180,E1 -22408.909,E2 -22408.909} C_VEL
LIN {X 0,Y 184.73,Z 602.292,A -85,B 0,C 180,E1 -22411.09,E2 -22411.09} C_VEL
LIN {X 0,Y 184.726,Z 597.208,A -85,B 0,C 180,E1 -22414.364,E2 -22414.364} C_VEL
LIN {X 0,Y 184.893,Z 591.712,A -85,B 0,C 180,E1 -22417.223,E2 -22417.223} C_VEL
LIN {X 0,Y 184.94,Z 588.92,A -85,B 0,C 180,E1 -22418.478,E2 -22418.478} C_VEL
LIN {X 0,Y 184.448,Z 585.325,A -85,B 0,C 180,E1 -22419.925,E2 -22419.925} C_VEL
LIN {X 0,Y 182.03,Z 578.729,A -85,B 0,C 180,E1 -22422.12,E2 -22422.12} C_VEL
LIN {X 0,Y 179.795,Z 571.585,A -85,B 0,C 180,E1 -22424.215,E2 -22424.215} C_VEL
LIN {X 0,Y 179.627,Z 567.124,A -85,B 0,C 180,E1 -22425.47,E2 -22425.47} C_VEL
LIN {X 0,Y 180.695,Z 557.936,A -85,B 0,C 180,E1 -22427.836,E2 -22427.836} C_VEL
LIN {X 0,Y 179.395,Z 546.202,A -85,B 0,C 180,E1 -22430.248,E2 -22430.248} C_VEL
LIN {X 0,Y 178.241,Z 532.978,A -85,B 0,C 180,E1 -22432.456,E2 -22432.456} C_VEL
LIN {X 0,Y 177.578,Z 520.158,A -85,B 0,C 180,E1 -22434.174,E2 -22434.174} C_VEL
LIN {X 0,Y 177.432,Z 510.941,A -85,B 0,C 180,E1 -22435.214,E2 -22435.214} C_VEL
LIN {X 0,Y 178.609,Z 506.198,A -85,B 0,C 180,E1 -22440.766,E2 -22440.766} C_VEL
LIN {X 0,Y 179.899,Z 501.771,A -85,B 0,C 180,E1 -22445.873,E2 -22445.873} C_VEL
LIN {X 0,Y 179.941,Z 499.368,A -85,B 0,C 180,E1 -22448.676,E2 -22448.676} C_VEL
LIN {X 0,Y 178.932,Z 494.275,A -85,B 0,C 180,E1 -22454.831,E2 -22454.831} C_VEL
LIN {X 0,Y 178.668,Z 494.229,A -85,B 0,C 180,E1 -22458.363,E2 -22458.363} C_VEL
LIN {X 0,Y 178.468,Z 494.25,A -85,B 0,C 180,E1 -22463.794,E2 -22463.794} C_VEL
LIN {X 0,Y 178.49,Z 494.252,A -85,B 0,C 180,E1 -22466.548,E2 -22466.548} C_VEL
LIN {X 0,Y 178.522,Z 494.245,A -85,B 0,C 180,E1 -22470.007,E2 -22470.007} C_VEL
LIN {X 0,Y 178.535,Z 494.246,A -85,B 0,C 180,E1 -22474.876,E2 -22474.876} C_VEL
LIN {X 0,Y 178.639,Z 494.229,A -85,B 0,C 180,E1 -22480.77,E2 -22480.77} C_VEL
LIN {X 0,Y 178.676,Z 494.227,A -85,B 0,C 180,E1 -22484.018,E2 -22484.018} C_VEL
LIN {X 0,Y 178.896,Z 494.196,A -85,B 0,C 180,E1 -22489.154,E2 -22489.154} C_VEL
LIN {X 0,Y 178.935,Z 494.195,A -85,B 0,C 180,E1 -22493.233,E2 -22493.233} C_VEL
LIN {X 0,Y 179.156,Z 494.162,A -85,B 0,C 180,E1 -22497.752,E2 -22497.752} C_VEL
LIN {X 0,Y 179.372,Z 494.139,A -85,B 0,C 180,E1 -22500,E2 -22500} C_VEL
LIN {X 0,Y 178.878,Z 494.202,A -85,B 0,C 180,E1 -22504.507,E2 -22504.507} C_VEL
LIN {X 0,Y 178.98,Z 494.189,A -85,B 0,C 180,E1 -22509.037,E2 -22509.037} C_VEL
LIN {X 0,Y 178.683,Z 494.224,A -85,B 0,C 180,E1 -22513.651,E2 -22513.651} C_VEL
LIN {X 0,Y 178.625,Z 494.233,A -85,B 0,C 180,E1 -22519.217,E2 -22519.217} C_VEL
LIN {X 0,Y 178.536,Z 494.242,A -85,B 0,C 180,E1 -22525.125,E2 -22525.125} C_VEL
LIN {X 0,Y 178.481,Z 494.25,A -85,B 0,C 180,E1 -22530.791,E2 -22530.791} C_VEL
LIN {X 0,Y 178.487,Z 494.249,A -85,B 0,C 180,E1 -22534.22,E2 -22534.22} C_VEL
LIN {X 0,Y 178.397,Z 494.261,A -85,B 0,C 180,E1 -22539.075,E2 -22539.075} C_VEL
LIN {X 0,Y 178.4,Z 494.258,A -85,B 0,C 180,E1 -22542.045,E2 -22542.045} C_VEL
LIN {X 0,Y 178.403,Z 494.261,A -85,B 0,C 180,E1 -22545.162,E2 -22545.162} C_VEL
LIN {X 0,Y 178.413,Z 494.259,A -85,B 0,C 180,E1 -22548.457,E2 -22548.457} C_VEL
LIN {X 0,Y 178.466,Z 494.251,A -85,B 0,C 180,E1 -22551.963,E2 -22551.963} C_VEL
LIN {X 0,Y 178.494,Z 494.249,A -85,B 0,C 180,E1 -22556.548,E2 -22556.548} C_VEL
LIN {X 0,Y 178.525,Z 494.242,A -85,B 0,C 180,E1 -22560.007,E2 -22560.007} C_VEL
LIN {X 0,Y 178.537,Z 494.244,A -85,B 0,C 180,E1 -22564.876,E2 -22564.876} C_VEL
LIN {X 0,Y 178.626,Z 494.233,A -85,B 0,C 180,E1 -22570.784,E2 -22570.784} C_VEL
LIN {X 0,Y 178.662,Z 494.225,A -85,B 0,C 180,E1 -22576.348,E2 -22576.348} C_VEL
LIN {X 0,Y 178.912,Z 494.198,A -85,B 0,C 180,E1 -22580.96,E2 -22580.96} C_VEL
LIN {X 0,Y 179.154,Z 494.167,A -85,B 0,C 180,E1 -22587.752,E2 -22587.752} C_VEL
LIN {X 0,Y 179.374,Z 494.143,A -85,B 0,C 180,E1 -22590,E2 -22590} C_VEL
LIN {X 0,Y 178.872,Z 494.199,A -85,B 0,C 180,E1 -22594.507,E2 -22594.507} C_VEL
LIN {X 0,Y 178.915,Z 494.197,A -85,B 0,C 180,E1 -22599.04,E2 -22599.04} C_VEL
LIN {X 0,Y 178.663,Z 494.225,A -85,B 0,C 180,E1 -22603.652,E2 -22603.652} C_VEL
LIN {X 0,Y 178.627,Z 494.233,A -85,B 0,C 180,E1 -22609.217,E2 -22609.217} C_VEL
LIN {X 0,Y 178.538,Z 494.244,A -85,B 0,C 180,E1 -22615.124,E2 -22615.124} C_VEL
LIN {X 0,Y 178.482,Z 494.246,A -85,B 0,C 180,E1 -22620.79,E2 -22620.79} C_VEL
LIN {X 0,Y 178.499,Z 494.25,A -85,B 0,C 180,E1 -22624.225,E2 -22624.225} C_VEL
LIN {X 0,Y 178.422,Z 494.255,A -85,B 0,C 180,E1 -22629.068,E2 -22629.068} C_VEL
LIN {X 0,Y 178.406,Z 494.262,A -85,B 0,C 180,E1 -22632.043,E2 -22632.043} C_VEL
LIN {X 0,Y 178.401,Z 494.262,A -85,B 0,C 180,E1 -22635.162,E2 -22635.162} C_VEL
LIN {X 0,Y 178.398,Z 494.257,A -85,B 0,C 180,E1 -22638.462,E2 -22638.462} C_VEL
LIN {X 0,Y 178.321,Z 494.273,A -85,B 0,C 180,E1 -22642.022,E2 -22642.022} C_VEL
LIN {X 0,Y 178.134,Z 494.29,A -85,B 0,C 180,E1 -22646.471,E2 -22646.471} C_VEL
LIN {X 0,Y 177.572,Z 494.367,A -85,B 0,C 180,E1 -22651.644,E2 -22651.644} C_VEL
LIN {X 0,Y 177.339,Z 494.395,A -85,B 0,C 180,E1 -22655.597,E2 -22655.597} C_VEL
LIN {X 0,Y 179.65,Z 508.895,A -85,B 0,C 180,E1 -22657.437,E2 -22657.437} C_VEL
LIN {X 0,Y 182.067,Z 522.863,A -85,B 0,C 180,E1 -22659.67,E2 -22659.67} C_VEL
LIN {X 0,Y 180.948,Z 532.82,A -85,B 0,C 180,E1 -22661.604,E2 -22661.604} C_VEL
LIN {X 0,Y 179.64,Z 543.545,A -85,B 0,C 180,E1 -22664.106,E2 -22664.106} C_VEL
LIN {X 0,Y 178.336,Z 555.333,A -85,B 0,C 180,E1 -22667.481,E2 -22667.481} C_VEL
LIN {X 0,Y 177.336,Z 564.888,A -85,B 0,C 180,E1 -22670.878,E2 -22670.878} C_VEL
LIN {X 0,Y 176.758,Z 573.486,A -85,B 0,C 180,E1 -22674.643,E2 -22674.643} C_VEL
LIN {X 0,Y 176.602,Z 579.306,A -85,B 0,C 180,E1 -22677.719,E2 -22677.719} C_VEL
LIN {X 0,Y 176.582,Z 584.678,A -85,B 0,C 180,E1 -22681.14,E2 -22681.14} C_VEL
LIN {X 0,Y 177.213,Z 590.295,A -85,B 0,C 180,E1 -22685.69,E2 -22685.69} C_VEL
LIN {X 0,Y 178.463,Z 594.299,A -85,B 0,C 180,E1 -22690.093,E2 -22690.093} C_VEL
LIN {X 0,Y 180.387,Z 596.57,A -85,B 0,C 180,E1 -22693.518,E2 -22693.518} C_VEL
LIN {X 0,Y 183.773,Z 598.345,A -85,B 0,C 180,E1 -22697.815,E2 -22697.815} C_VEL
LIN {X 0,Y 188.351,Z 598.849,A -85,B 0,C 180,E1 -22701.909,E2 -22701.909} C_VEL
LIN {X 0,Y 194.01,Z 598.131,A -85,B 0,C 180,E1 -22705.766,E2 -22705.766} C_VEL
LIN {X 0,Y 200.712,Z 596.189,A -85,B 0,C 180,E1 -22709.355,E2 -22709.355} C_VEL
LIN {X 0,Y 208.411,Z 593.016,A -85,B 0,C 180,E1 -22712.653,E2 -22712.653} C_VEL
LIN {X 0,Y 217.045,Z 588.434,A -85,B 0,C 180,E1 -22715.651,E2 -22715.651} C_VEL
LIN {X 0,Y 221.601,Z 585.663,A -85,B 0,C 180,E1 -22717.055,E2 -22717.055} C_VEL
LIN {X 0,Y 222.547,Z 584.955,A -85,B 0,C 180,E1 -22717.861,E2 -22717.861} C_VEL
LIN {X 0,Y 222.969,Z 584.536,A -85,B 0,C 180,E1 -22719.08,E2 -22719.08} C_VEL
LIN {X 0,Y 223.447,Z 584.168,A -85,B 0,C 180,E1 -22721.338,E2 -22721.338} C_VEL
LIN {X 0,Y 223.427,Z 584.613,A -85,B 0,C 180,E1 -22723.79,E2 -22723.79} C_VEL
LIN {X 0,Y 222.141,Z 586.545,A -85,B 0,C 180,E1 -22726.691,E2 -22726.691} C_VEL
LIN {X 0,Y 219.21,Z 589.583,A -85,B 0,C 180,E1 -22728.91,E2 -22728.91} C_VEL
LIN {X 0,Y 216.401,Z 592.329,A -85,B 0,C 180,E1 -22730.706,E2 -22730.706} C_VEL
LIN {X 0,Y 214.829,Z 593.736,A -85,B 0,C 180,E1 -22731.568,E2 -22731.568} C_VEL
LIN {X 0,Y 210.767,Z 596.735,A -85,B 0,C 180,E1 -22733.115,E2 -22733.115} C_VEL
LIN {X 0,Y 202.385,Z 602.11,A -85,B 0,C 180,E1 -22736.247,E2 -22736.247} C_VEL
LIN {X 0,Y 195.051,Z 606.236,A -85,B 0,C 180,E1 -22739.705,E2 -22739.705} C_VEL
LIN {X 0,Y 188.858,Z 609.187,A -85,B 0,C 180,E1 -22743.477,E2 -22743.477} C_VEL
LIN {X 0,Y 183.968,Z 611.005,A -85,B 0,C 180,E1 -22747.541,E2 -22747.541} C_VEL
LIN {X 0,Y 180.273,Z 611.661,A -85,B 0,C 180,E1 -22751.827,E2 -22751.827} C_VEL
LIN {X 0,Y 177.956,Z 611.161,A -85,B 0,C 180,E1 -22756.293,E2 -22756.293} C_VEL
LIN {X 0,Y 176.974,Z 609.456,A -85,B 0,C 180,E1 -22760.86,E2 -22760.86} C_VEL
LIN {X 0,Y 177.061,Z 606.464,A -85,B 0,C 180,E1 -22765.447,E2 -22765.447} C_VEL
LIN {X 0,Y 177.7,Z 603.2,A -85,B 0,C 180,E1 -22768.867,E2 -22768.867} C_VEL
LIN {X 0,Y 177.847,Z 600.379,A -85,B 0,C 180,E1 -22771.132,E2 -22771.132} C_VEL
LIN {X 0,Y 177.847,Z 595.082,A -85,B 0,C 180,E1 -22774.533,E2 -22774.533} C_VEL
LIN {X 0,Y 177.981,Z 589.199,A -85,B 0,C 180,E1 -22777.54,E2 -22777.54} C_VEL
LIN {X 0,Y 178.357,Z 581.618,A -85,B 0,C 180,E1 -22780.73,E2 -22780.73} C_VEL
LIN {X 0,Y 178.989,Z 573.31,A -85,B 0,C 180,E1 -22783.626,E2 -22783.626} C_VEL
LIN {X 0,Y 179.627,Z 567.124,A -85,B 0,C 180,E1 -22785.47,E2 -22785.47} C_VEL
LIN {X 0,Y 179.589,Z 564.167,A -85,B 0,C 180,E1 -22786.265,E2 -22786.265} C_VEL
LIN {X 0,Y 178.922,Z 561.056,A -85,B 0,C 180,E1 -22787.011,E2 -22787.011} C_VEL
LIN {X 0,Y 176.47,Z 554.813,A -85,B 0,C 180,E1 -22788.373,E2 -22788.373} C_VEL
LIN {X 0,Y 172.5,Z 544.892,A -85,B 0,C 180,E1 -22790.307,E2 -22790.307} C_VEL
LIN {X 0,Y 171.839,Z 541.324,A -85,B 0,C 180,E1 -22790.961,E2 -22790.961} C_VEL
LIN {X 0,Y 170.772,Z 527.605,A -85,B 0,C 180,E1 -22793.175,E2 -22793.175} C_VEL
LIN {X 0,Y 170.3,Z 513.843,A -85,B 0,C 180,E1 -22794.911,E2 -22794.911} C_VEL
LIN {X 0,Y 170.349,Z 510.592,A -85,B 0,C 180,E1 -22795.297,E2 -22795.297} C_VEL
LIN {X 0,Y 171.796,Z 505.012,A -85,B 0,C 180,E1 -22802.128,E2 -22802.128} C_VEL
LIN {X 0,Y 172.664,Z 502.217,A -85,B 0,C 180,E1 -22805.505,E2 -22805.505} C_VEL
LIN {X 0,Y 172.928,Z 500.524,A -85,B 0,C 180,E1 -22807.562,E2 -22807.562} C_VEL
LIN {X 0,Y 172.462,Z 498.006,A -85,B 0,C 180,E1 -22810.694,E2 -22810.694} C_VEL
LIN {X 0,Y 171.903,Z 495.073,A -85,B 0,C 180,E1 -22814.494,E2 -22814.494} C_VEL
LIN {X 0,Y 171.548,Z 495.116,A -85,B 0,C 180,E1 -22819.043,E2 -22819.043} C_VEL
LIN {X 0,Y 171.454,Z 495.123,A -85,B 0,C 180,E1 -22822.059,E2 -22822.059} C_VEL
LIN {X 0,Y 171.418,Z 495.131,A -85,B 0,C 180,E1 -22827.793,E2 -22827.793} C_VEL
LIN {X 0,Y 171.448,Z 495.125,A -85,B 0,C 180,E1 -22830.534,E2 -22830.534} C_VEL
LIN {X 0,Y 171.459,Z 495.126,A -85,B 0,C 180,E1 -22835.802,E2 -22835.802} C_VEL
LIN {X 0,Y 171.596,Z 495.107,A -85,B 0,C 180,E1 -22840.874,E2 -22840.874} C_VEL
LIN {X 0,Y 171.614,Z 495.107,A -85,B 0,C 180,E1 -22845.776,E2 -22845.776} C_VEL
LIN {X 0,Y 171.911,Z 495.069,A -85,B 0,C 180,E1 -22850.589,E2 -22850.589} C_VEL
LIN {X 0,Y 171.827,Z 495.079,A -85,B 0,C 180,E1 -22855.308,E2 -22855.308} C_VEL
LIN {X 0,Y 172.335,Z 495.016,A -85,B 0,C 180,E1 -22860,E2 -22860} C_VEL
LIN {X 0,Y 171.828,Z 495.079,A -85,B 0,C 180,E1 -22864.693,E2 -22864.693} C_VEL
LIN {X 0,Y 171.912,Z 495.069,A -85,B 0,C 180,E1 -22869.412,E2 -22869.412} C_VEL
LIN {X 0,Y 171.596,Z 495.107,A -85,B 0,C 180,E1 -22874.226,E2 -22874.226} C_VEL
LIN {X 0,Y 171.546,Z 495.115,A -85,B 0,C 180,E1 -22879.563,E2 -22879.563} C_VEL
LIN {X 0,Y 171.471,Z 495.122,A -85,B 0,C 180,E1 -22885.617,E2 -22885.617} C_VEL
LIN {X 0,Y 171.444,Z 495.127,A -85,B 0,C 180,E1 -22890.588,E2 -22890.588} C_VEL
LIN {X 0,Y 171.394,Z 495.133,A -85,B 0,C 180,E1 -22895.035,E2 -22895.035} C_VEL
LIN {X 0,Y 171.359,Z 495.138,A -85,B 0,C 180,E1 -22898.808,E2 -22898.808} C_VEL
LIN {X 0,Y 171.326,Z 495.143,A -85,B 0,C 180,E1 -22904.216,E2 -22904.216} C_VEL
LIN {X 0,Y 171.347,Z 495.137,A -85,B 0,C 180,E1 -22908.985,E2 -22908.985} C_VEL
LIN {X 0,Y 171.416,Z 495.13,A -85,B 0,C 180,E1 -22912.049,E2 -22912.049} C_VEL
LIN {X 0,Y 171.413,Z 495.132,A -85,B 0,C 180,E1 -22915.087,E2 -22915.087} C_VEL
LIN {X 0,Y 171.452,Z 495.126,A -85,B 0,C 180,E1 -22920.535,E2 -22920.535} C_VEL
LIN {X 0,Y 171.461,Z 495.127,A -85,B 0,C 180,E1 -22925.802,E2 -22925.802} C_VEL
LIN {X 0,Y 171.583,Z 495.11,A -85,B 0,C 180,E1 -22930.872,E2 -22930.872} C_VEL
LIN {X 0,Y 171.58,Z 495.11,A -85,B 0,C 180,E1 -22935.773,E2 -22935.773} C_VEL
LIN {X 0,Y 171.849,Z 495.078,A -85,B 0,C 180,E1 -22940.585,E2 -22940.585} C_VEL
LIN {X 0,Y 171.813,Z 495.078,A -85,B 0,C 180,E1 -22945.308,E2 -22945.308} C_VEL
LIN {X 0,Y 172.336,Z 495.02,A -85,B 0,C 180,E1 -22950,E2 -22950} C_VEL
LIN {X 0,Y 171.82,Z 495.077,A -85,B 0,C 180,E1 -22954.693,E2 -22954.693} C_VEL
LIN {X 0,Y 171.852,Z 495.078,A -85,B 0,C 180,E1 -22959.415,E2 -22959.415} C_VEL
LIN {X 0,Y 171.581,Z 495.11,A -85,B 0,C 180,E1 -22964.227,E2 -22964.227} C_VEL
LIN {X 0,Y 171.548,Z 495.116,A -85,B 0,C 180,E1 -22969.563,E2 -22969.563} C_VEL
LIN {X 0,Y 171.473,Z 495.125,A -85,B 0,C 180,E1 -22975.617,E2 -22975.617} C_VEL
LIN {X 0,Y 171.445,Z 495.122,A -85,B 0,C 180,E1 -22980.587,E2 -22980.587} C_VEL
LIN {X 0,Y 171.41,Z 495.132,A -85,B 0,C 180,E1 -22985.031,E2 -22985.031} C_VEL
LIN {X 0,Y 171.383,Z 495.131,A -85,B 0,C 180,E1 -22988.817,E2 -22988.817} C_VEL
LIN {X 0,Y 171.33,Z 495.143,A -85,B 0,C 180,E1 -22994.215,E2 -22994.215} C_VEL
LIN {X 0,Y 171.324,Z 495.138,A -85,B 0,C 180,E1 -22998.977,E2 -22998.977} C_VEL
LIN {X 0,Y 171.274,Z 495.151,A -85,B 0,C 180,E1 -23002.011,E2 -23002.011} C_VEL
LIN {X 0,Y 171.093,Z 495.171,A -85,B 0,C 180,E1 -23005.24,E2 -23005.24} C_VEL
LIN {X 0,Y 170.654,Z 495.226,A -85,B 0,C 180,E1 -23010.383,E2 -23010.383} C_VEL
LIN {X 0,Y 170.324,Z 495.468,A -85,B 0,C 180,E1 -23015.593,E2 -23015.593} C_VEL
LIN {X 0,Y 172.647,Z 509.973,A -85,B 0,C 180,E1 -23017.518,E2 -23017.518} C_VEL
LIN {X 0,Y 174.945,Z 523.177,A -85,B 0,C 180,E1 -23019.727,E2 -23019.727} C_VEL
LIN {X 0,Y 173.621,Z 534.429,A -85,B 0,C 180,E1 -23022.021,E2 -23022.021} C_VEL
LIN {X 0,Y 172.314,Z 544.889,A -85,B 0,C 180,E1 -23024.626,E2 -23024.626} C_VEL
LIN {X 0,Y 171.059,Z 556.368,A -85,B 0,C 180,E1 -23028.145,E2 -23028.145} C_VEL
LIN {X 0,Y 170.202,Z 565.751,A -85,B 0,C 180,E1 -23031.691,E2 -23031.691} C_VEL
LIN {X 0,Y 169.646,Z 574.743,A -85,B 0,C 180,E1 -23035.842,E2 -23035.842} C_VEL
LIN {X 0,Y 169.546,Z 579.975,A -85,B 0,C 180,E1 -23038.812,E2 -23038.812} C_VEL
LIN {X 0,Y 169.659,Z 585.247,A -85,B 0,C 180,E1 -23042.374,E2 -23042.374} C_VEL
LIN {X 0,Y 170.189,Z 589.587,A -85,B 0,C 180,E1 -23045.925,E2 -23045.925} C_VEL
LIN {X 0,Y 171.392,Z 593.668,A -85,B 0,C 180,E1 -23050.218,E2 -23050.218} C_VEL
LIN {X 0,Y 173.493,Z 596.452,A -85,B 0,C 180,E1 -23054.066,E2 -23054.066} C_VEL
LIN {X 0,Y 177.03,Z 598.582,A -85,B 0,C 180,E1 -23058.517,E2 -23058.517} C_VEL
LIN {X 0,Y 181.831,Z 599.493,A -85,B 0,C 180,E1 -23062.737,E2 -23062.737} C_VEL
LIN {X 0,Y 187.725,Z 599.195,A -85,B 0,C 180,E1 -23066.696,E2 -23066.696} C_VEL
LIN {X 0,Y 194.702,Z 597.691,A -85,B 0,C 180,E1 -23070.354,E2 -23070.354} C_VEL
LIN {X 0,Y 203.401,Z 594.628,A -85,B 0,C 180,E1 -23073.977,E2 -23073.977} C_VEL
LIN {X 0,Y 211.567,Z 590.912,A -85,B 0,C 180,E1 -23076.722,E2 -23076.722} C_VEL
LIN {X 0,Y 216.251,Z 588.419,A -85,B 0,C 180,E1 -23078.133,E2 -23078.133} C_VEL
LIN {X 0,Y 216.715,Z 588.153,A -85,B 0,C 180,E1 -23078.893,E2 -23078.893} C_VEL
LIN {X 0,Y 217.091,Z 587.914,A -85,B 0,C 180,E1 -23080.351,E2 -23080.351} C_VEL
LIN {X 0,Y 217.317,Z 588.07,A -85,B 0,C 180,E1 -23082.776,E2 -23082.776} C_VEL
LIN {X 0,Y 216.503,Z 589.368,A -85,B 0,C 180,E1 -23085.574,E2 -23085.574} C_VEL
LIN {X 0,Y 215.339,Z 590.507,A -85,B 0,C 180,E1 -23086.735,E2 -23086.735} C_VEL
LIN {X 0,Y 211.077,Z 594.171,A -85,B 0,C 180,E1 -23089.513,E2 -23089.513} C_VEL
LIN {X 0,Y 209.432,Z 595.412,A -85,B 0,C 180,E1 -23090.387,E2 -23090.387} C_VEL
LIN {X 0,Y 205.223,Z 598.175,A -85,B 0,C 180,E1 -23091.944,E2 -23091.944} C_VEL
LIN {X 0,Y 196.584,Z 602.994,A -85,B 0,C 180,E1 -23095.109,E2 -23095.109} C_VEL
LIN {X 0,Y 188.966,Z 606.66,A -85,B 0,C 180,E1 -23098.621,E2 -23098.621} C_VEL
LIN {X 0,Y 182.538,Z 609.201,A -85,B 0,C 180,E1 -23102.482,E2 -23102.482} C_VEL
LIN {X 0,Y 177.425,Z 610.636,A -85,B 0,C 180,E1 -23106.664,E2 -23106.664} C_VEL
LIN {X 0,Y 173.554,Z 610.95,A -85,B 0,C 180,E1 -23111.097,E2 -23111.097} C_VEL
LIN {X 0,Y 171.103,Z 610.135,A -85,B 0,C 180,E1 -23115.732,E2 -23115.732} C_VEL
LIN {X 0,Y 170.049,Z 608.168,A -85,B 0,C 180,E1 -23120.484,E2 -23120.484} C_VEL
LIN {X 0,Y 170.175,Z 604.85,A -85,B 0,C 180,E1 -23125.262,E2 -23125.262} C_VEL
LIN {X 0,Y 170.836,Z 601.43,A -85,B 0,C 180,E1 -23128.821,E2 -23128.821} C_VEL
LIN {X 0,Y 170.953,Z 598.391,A -85,B 0,C 180,E1 -23131.178,E2 -23131.178} C_VEL
LIN {X 0,Y 170.99,Z 592.764,A -85,B 0,C 180,E1 -23134.715,E2 -23134.715} C_VEL
LIN {X 0,Y 171.098,Z 586.494,A -85,B 0,C 180,E1 -23137.901,E2 -23137.901} C_VEL
LIN {X 0,Y 171.528,Z 578.53,A -85,B 0,C 180,E1 -23141.222,E2 -23141.222} C_VEL
LIN {X 0,Y 172.407,Z 568.015,A -85,B 0,C 180,E1 -23144.76,E2 -23144.76} C_VEL
LIN {X 0,Y 173.59,Z 557.239,A -85,B 0,C 180,E1 -23147.677,E2 -23147.677} C_VEL
LIN {X 0,Y 172.255,Z 545.334,A -85,B 0,C 180,E1 -23150.216,E2 -23150.216} C_VEL
LIN {X 0,Y 171.839,Z 541.324,A -85,B 0,C 180,E1 -23150.961,E2 -23150.961} C_VEL
LIN {X 0,Y 170.656,Z 536.186,A -85,B 0,C 180,E1 -23151.869,E2 -23151.869} C_VEL
LIN {X 0,Y 167.083,Z 527.742,A -85,B 0,C 180,E1 -23153.189,E2 -23153.189} C_VEL
LIN {X 0,Y 163.859,Z 519.028,A -85,B 0,C 180,E1 -23154.357,E2 -23154.357} C_VEL
LIN {X 0,Y 163.217,Z 513.485,A -85,B 0,C 180,E1 -23155,E2 -23155} C_VEL
LIN {X 0,Y 163.291,Z 510.218,A -85,B 0,C 180,E1 -23155.369,E2 -23155.369} C_VEL
LIN {X 0,Y 164.477,Z 505.651,A -85,B 0,C 180,E1 -23161.286,E2 -23161.286} C_VEL
LIN {X 0,Y 165.657,Z 501.73,A -85,B 0,C 180,E1 -23166.286,E2 -23166.286} C_VEL
LIN {X 0,Y 165.797,Z 500.441,A -85,B 0,C 180,E1 -23167.926,E2 -23167.926} C_VEL
LIN {X 0,Y 164.986,Z 496.593,A -85,B 0,C 180,E1 -23172.966,E2 -23172.966} C_VEL
LIN {X 0,Y 164.888,Z 495.946,A -85,B 0,C 180,E1 -23174.158,E2 -23174.158} C_VEL
LIN {X 0,Y 164.443,Z 496,A -85,B 0,C 180,E1 -23180.29,E2 -23180.29} C_VEL
LIN {X 0,Y 164.333,Z 496.014,A -85,B 0,C 180,E1 -23186.223,E2 -23186.223} C_VEL
LIN {X 0,Y 164.389,Z 496.005,A -85,B 0,C 180,E1 -23189.135,E2 -23189.135} C_VEL
LIN {X 0,Y 164.417,Z 496.005,A -85,B 0,C 180,E1 -23194.694,E2 -23194.694} C_VEL
LIN {X 0,Y 164.486,Z 495.991,A -85,B 0,C 180,E1 -23200.05,E2 -23200.05} C_VEL
LIN {X 0,Y 164.56,Z 495.986,A -85,B 0,C 180,E1 -23205.153,E2 -23205.153} C_VEL
LIN {X 0,Y 164.854,Z 495.945,A -85,B 0,C 180,E1 -23210.182,E2 -23210.182} C_VEL
LIN {X 0,Y 164.863,Z 495.95,A -85,B 0,C 180,E1 -23212.653,E2 -23212.653} C_VEL
LIN {X 0,Y 165.052,Z 495.919,A -85,B 0,C 180,E1 -23217.56,E2 -23217.56} C_VEL
LIN {X 0,Y 165.297,Z 495.892,A -85,B 0,C 180,E1 -23220,E2 -23220} C_VEL
LIN {X 0,Y 164.843,Z 495.945,A -85,B 0,C 180,E1 -23227.115,E2 -23227.115} C_VEL
LIN {X 0,Y 164.781,Z 495.958,A -85,B 0,C 180,E1 -23231.198,E2 -23231.198} C_VEL
LIN {X 0,Y 164.487,Z 495.993,A -85,B 0,C 180,E1 -23237.403,E2 -23237.403} C_VEL
LIN {X 0,Y 164.475,Z 495.997,A -85,B 0,C 180,E1 -23239.99,E2 -23239.99} C_VEL
LIN {X 0,Y 164.395,Z 496.005,A -85,B 0,C 180,E1 -23246.135,E2 -23246.135} C_VEL
LIN {X 0,Y 164.377,Z 496.006,A -85,B 0,C 180,E1 -23251.229,E2 -23251.229} C_VEL
LIN {X 0,Y 164.296,Z 496.019,A -85,B 0,C 180,E1 -23256.79,E2 -23256.79} C_VEL
LIN {X 0,Y 164.293,Z 496.019,A -85,B 0,C 180,E1 -23259.917,E2 -23259.917} C_VEL
LIN {X 0,Y 164.281,Z 496.018,A -85,B 0,C 180,E1 -23263.342,E2 -23263.342} C_VEL
LIN {X 0,Y 164.294,Z 496.019,A -85,B 0,C 180,E1 -23266.809,E2 -23266.809} C_VEL
LIN {X 0,Y 164.307,Z 496.013,A -85,B 0,C 180,E1 -23270.348,E2 -23270.348} C_VEL
LIN {X 0,Y 164.346,Z 496.014,A -85,B 0,C 180,E1 -23274.343,E2 -23274.343} C_VEL
LIN {X 0,Y 164.394,Z 496,A -85,B 0,C 180,E1 -23279.136,E2 -23279.136} C_VEL
LIN {X 0,Y 164.419,Z 496.003,A -85,B 0,C 180,E1 -23284.695,E2 -23284.695} C_VEL
LIN {X 0,Y 164.487,Z 495.994,A -85,B 0,C 180,E1 -23290.051,E2 -23290.051} C_VEL
LIN {X 0,Y 164.528,Z 495.987,A -85,B 0,C 180,E1 -23295.15,E2 -23295.15} C_VEL
LIN {X 0,Y 164.77,Z 495.962,A -85,B 0,C 180,E1 -23300.177,E2 -23300.177} C_VEL
LIN {X 0,Y 164.83,Z 495.951,A -85,B 0,C 180,E1 -23302.651,E2 -23302.651} C_VEL
LIN {X 0,Y 165.049,Z 495.923,A -85,B 0,C 180,E1 -23307.56,E2 -23307.56} C_VEL
LIN {X 0,Y 165.299,Z 495.896,A -85,B 0,C 180,E1 -23310,E2 -23310} C_VEL
LIN {X 0,Y 164.768,Z 495.955,A -85,B 0,C 180,E1 -23314.894,E2 -23314.894} C_VEL
LIN {X 0,Y 164.835,Z 495.951,A -85,B 0,C 180,E1 -23317.349,E2 -23317.349} C_VEL
LIN {X 0,Y 164.706,Z 495.966,A -85,B 0,C 180,E1 -23321.062,E2 -23321.062} C_VEL
LIN {X 0,Y 164.488,Z 495.995,A -85,B 0,C 180,E1 -23327.403,E2 -23327.403} C_VEL
LIN {X 0,Y 164.477,Z 495.995,A -85,B 0,C 180,E1 -23329.989,E2 -23329.989} C_VEL
LIN {X 0,Y 164.397,Z 496.007,A -85,B 0,C 180,E1 -23336.134,E2 -23336.134} C_VEL
LIN {X 0,Y 164.379,Z 496.003,A -85,B 0,C 180,E1 -23341.228,E2 -23341.228} C_VEL
LIN {X 0,Y 164.316,Z 496.015,A -85,B 0,C 180,E1 -23346.784,E2 -23346.784} C_VEL
LIN {X 0,Y 164.303,Z 496.014,A -85,B 0,C 180,E1 -23349.913,E2 -23349.913} C_VEL
LIN {X 0,Y 164.282,Z 496.021,A -85,B 0,C 180,E1 -23353.342,E2 -23353.342} C_VEL
LIN {X 0,Y 164.265,Z 496.02,A -85,B 0,C 180,E1 -23356.799,E2 -23356.799} C_VEL
LIN {X 0,Y 164.227,Z 496.026,A -85,B 0,C 180,E1 -23360.381,E2 -23360.381} C_VEL
LIN {X 0,Y 164.056,Z 496.047,A -85,B 0,C 180,E1 -23364.484,E2 -23364.484} C_VEL
LIN {X 0,Y 163.688,Z 496.092,A -85,B 0,C 180,E1 -23369.173,E2 -23369.173} C_VEL
LIN {X 0,Y 163.277,Z 496.314,A -85,B 0,C 180,E1 -23375.572,E2 -23375.572} C_VEL
LIN {X 0,Y 165.54,Z 510.484,A -85,B 0,C 180,E1 -23377.536,E2 -23377.536} C_VEL
LIN {X 0,Y 167.784,Z 523.661,A -85,B 0,C 180,E1 -23379.833,E2 -23379.833} C_VEL
LIN {X 0,Y 166.351,Z 535.773,A -85,B 0,C 180,E1 -23382.481,E2 -23382.481} C_VEL
LIN {X 0,Y 164.804,Z 548.016,A -85,B 0,C 180,E1 -23385.805,E2 -23385.805} C_VEL
LIN {X 0,Y 163.821,Z 557.295,A -85,B 0,C 180,E1 -23388.869,E2 -23388.869} C_VEL
LIN {X 0,Y 163.083,Z 566.595,A -85,B 0,C 180,E1 -23392.571,E2 -23392.571} C_VEL
LIN {X 0,Y 162.63,Z 575.371,A -85,B 0,C 180,E1 -23396.903,E2 -23396.903} C_VEL
LIN {X 0,Y 162.559,Z 582.409,A -85,B 0,C 180,E1 -23401.238,E2 -23401.238} C_VEL
LIN {X 0,Y 162.971,Z 587.325,A -85,B 0,C 180,E1 -23404.947,E2 -23404.947} C_VEL
LIN {X 0,Y 164.113,Z 592.434,A -85,B 0,C 180,E1 -23409.863,E2 -23409.863} C_VEL
LIN {X 0,Y 166.642,Z 596.208,A -85,B 0,C 180,E1 -23414.657,E2 -23414.657} C_VEL
LIN {X 0,Y 170.33,Z 598.733,A -85,B 0,C 180,E1 -23419.274,E2 -23419.274} C_VEL
LIN {X 0,Y 175.338,Z 600.033,A -85,B 0,C 180,E1 -23423.63,E2 -23423.63} C_VEL
LIN {X 0,Y 181.488,Z 600.117,A -85,B 0,C 180,E1 -23427.69,E2 -23427.69} C_VEL
LIN {X 0,Y 188.723,Z 599.027,A -85,B 0,C 180,E1 -23431.423,E2 -23431.423} C_VEL
LIN {X 0,Y 196.982,Z 596.764,A -85,B 0,C 180,E1 -23434.81,E2 -23434.81} C_VEL
LIN {X 0,Y 206.149,Z 593.261,A -85,B 0,C 180,E1 -23437.854,E2 -23437.854} C_VEL
LIN {X 0,Y 210.495,Z 591.308,A -85,B 0,C 180,E1 -23439.373,E2 -23439.373} C_VEL
LIN {X 0,Y 211.039,Z 591.25,A -85,B 0,C 180,E1 -23441.762,E2 -23441.762} C_VEL
LIN {X 0,Y 211.002,Z 591.471,A -85,B 0,C 180,E1 -23442.88,E2 -23442.88} C_VEL
LIN {X 0,Y 210.546,Z 592.119,A -85,B 0,C 180,E1 -23444.505,E2 -23444.505} C_VEL
LIN {X 0,Y 210.048,Z 592.677,A -85,B 0,C 180,E1 -23445.36,E2 -23445.36} C_VEL
LIN {X 0,Y 207.325,Z 594.702,A -85,B 0,C 180,E1 -23447.314,E2 -23447.314} C_VEL
LIN {X 0,Y 204.106,Z 597.002,A -85,B 0,C 180,E1 -23449.138,E2 -23449.138} C_VEL
LIN {X 0,Y 199.755,Z 599.456,A -85,B 0,C 180,E1 -23450.706,E2 -23450.706} C_VEL
LIN {X 0,Y 190.847,Z 603.786,A -85,B 0,C 180,E1 -23453.899,E2 -23453.899} C_VEL
LIN {X 0,Y 182.959,Z 606.984,A -85,B 0,C 180,E1 -23457.467,E2 -23457.467} C_VEL
LIN {X 0,Y 176.277,Z 609.099,A -85,B 0,C 180,E1 -23461.417,E2 -23461.417} C_VEL
LIN {X 0,Y 170.931,Z 610.149,A -85,B 0,C 180,E1 -23465.722,E2 -23465.722} C_VEL
LIN {X 0,Y 166.876,Z 610.104,A -85,B 0,C 180,E1 -23470.31,E2 -23470.31} C_VEL
LIN {X 0,Y 164.291,Z 608.98,A -85,B 0,C 180,E1 -23475.127,E2 -23475.127} C_VEL
LIN {X 0,Y 163.172,Z 606.687,A -85,B 0,C 180,E1 -23480.079,E2 -23480.079} C_VEL
LIN {X 0,Y 163.141,Z 605.111,A -85,B 0,C 180,E1 -23482.574,E2 -23482.574} C_VEL
LIN {X 0,Y 163.805,Z 600.81,A -85,B 0,C 180,E1 -23487.541,E2 -23487.541} C_VEL
LIN {X 0,Y 164.136,Z 597.964,A -85,B 0,C 180,E1 -23490,E2 -23490} C_VEL
LIN {X 0,Y 164.121,Z 592.488,A -85,B 0,C 180,E1 -23493.683,E2 -23493.683} C_VEL
LIN {X 0,Y 164.207,Z 585.513,A -85,B 0,C 180,E1 -23497.377,E2 -23497.377} C_VEL
LIN {X 0,Y 164.591,Z 577.466,A -85,B 0,C 180,E1 -23500.86,E2 -23500.86} C_VEL
LIN {X 0,Y 165.316,Z 568.256,A -85,B 0,C 180,E1 -23504.149,E2 -23504.149} C_VEL
LIN {X 0,Y 166.439,Z 557.784,A -85,B 0,C 180,E1 -23507.192,E2 -23507.192} C_VEL
LIN {X 0,Y 165.797,Z 550.726,A -85,B 0,C 180,E1 -23508.857,E2 -23508.857} C_VEL
LIN {X 0,Y 164.468,Z 537.808,A -85,B 0,C 180,E1 -23511.436,E2 -23511.436} C_VEL
LIN {X 0,Y 163.5,Z 524.445,A -85,B 0,C 180,E1 -23513.596,E2 -23513.596} C_VEL
LIN {X 0,Y 163.217,Z 513.485,A -85,B 0,C 180,E1 -23515,E2 -23515} C_VEL
LIN {X 0,Y 163.008,Z 511.12,A -85,B 0,C 180,E1 -23515.557,E2 -23515.557} C_VEL
LIN {X 0,Y 162.223,Z 509.11,A -85,B 0,C 180,E1 -23516.754,E2 -23516.754} C_VEL
LIN {X 0,Y 158.862,Z 504.98,A -85,B 0,C 180,E1 -23522.279,E2 -23522.279} C_VEL
LIN {X 0,Y 158.359,Z 502.47,A -85,B 0,C 180,E1 -23525.418,E2 -23525.418} C_VEL
LIN {X 0,Y 158.642,Z 500.298,A -85,B 0,C 180,E1 -23528.332,E2 -23528.332} C_VEL
LIN {X 0,Y 157.88,Z 496.82,A -85,B 0,C 180,E1 -23533.206,E2 -23533.206} C_VEL
LIN {X 0,Y 157.491,Z 496.866,A -85,B 0,C 180,E1 -23537.982,E2 -23537.982} C_VEL
LIN {X 0,Y 157.297,Z 496.888,A -85,B 0,C 180,E1 -23544.491,E2 -23544.491} C_VEL
LIN {X 0,Y 157.294,Z 496.891,A -85,B 0,C 180,E1 -23548.096,E2 -23548.096} C_VEL
LIN {X 0,Y 157.322,Z 496.886,A -85,B 0,C 180,E1 -23553.466,E2 -23553.466} C_VEL
LIN {X 0,Y 157.396,Z 496.873,A -85,B 0,C 180,E1 -23559.666,E2 -23559.666} C_VEL
LIN {X 0,Y 157.486,Z 496.869,A -85,B 0,C 180,E1 -23564.47,E2 -23564.47} C_VEL
LIN {X 0,Y 157.773,Z 496.826,A -85,B 0,C 180,E1 -23569.737,E2 -23569.737} C_VEL
LIN {X 0,Y 157.826,Z 496.825,A -85,B 0,C 180,E1 -23572.323,E2 -23572.323} C_VEL
LIN {X 0,Y 158.259,Z 496.769,A -85,B 0,C 180,E1 -23580,E2 -23580} C_VEL
LIN {X 0,Y 157.826,Z 496.82,A -85,B 0,C 180,E1 -23587.678,E2 -23587.678} C_VEL
LIN {X 0,Y 157.706,Z 496.839,A -85,B 0,C 180,E1 -23591.362,E2 -23591.362} C_VEL
LIN {X 0,Y 157.464,Z 496.863,A -85,B 0,C 180,E1 -23595.534,E2 -23595.534} C_VEL
LIN {X 0,Y 157.371,Z 496.881,A -85,B 0,C 180,E1 -23600.933,E2 -23600.933} C_VEL
LIN {X 0,Y 157.317,Z 496.889,A -85,B 0,C 180,E1 -23606.686,E2 -23606.686} C_VEL
LIN {X 0,Y 157.277,Z 496.889,A -85,B 0,C 180,E1 -23612.428,E2 -23612.428} C_VEL
LIN {X 0,Y 157.269,Z 496.896,A -85,B 0,C 180,E1 -23616.45,E2 -23616.45} C_VEL
LIN {X 0,Y 157.212,Z 496.897,A -85,B 0,C 180,E1 -23622.111,E2 -23622.111} C_VEL
LIN {X 0,Y 157.215,Z 496.901,A -85,B 0,C 180,E1 -23627.891,E2 -23627.891} C_VEL
LIN {X 0,Y 157.285,Z 496.891,A -85,B 0,C 180,E1 -23633.544,E2 -23633.544} C_VEL
LIN {X 0,Y 157.297,Z 496.887,A -85,B 0,C 180,E1 -23638.095,E2 -23638.095} C_VEL
LIN {X 0,Y 157.325,Z 496.887,A -85,B 0,C 180,E1 -23643.467,E2 -23643.467} C_VEL
LIN {X 0,Y 157.397,Z 496.875,A -85,B 0,C 180,E1 -23649.668,E2 -23649.668} C_VEL
LIN {X 0,Y 157.457,Z 496.869,A -85,B 0,C 180,E1 -23654.467,E2 -23654.467} C_VEL
LIN {X 0,Y 157.692,Z 496.841,A -85,B 0,C 180,E1 -23659.731,E2 -23659.731} C_VEL
LIN {X 0,Y 157.767,Z 496.832,A -85,B 0,C 180,E1 -23662.32,E2 -23662.32} C_VEL
LIN {X 0,Y 158.261,Z 496.773,A -85,B 0,C 180,E1 -23670,E2 -23670} C_VEL
LIN {X 0,Y 157.772,Z 496.832,A -85,B 0,C 180,E1 -23677.68,E2 -23677.68} C_VEL
LIN {X 0,Y 157.641,Z 496.846,A -85,B 0,C 180,E1 -23681.238,E2 -23681.238} C_VEL
LIN {X 0,Y 157.458,Z 496.869,A -85,B 0,C 180,E1 -23685.534,E2 -23685.534} C_VEL
LIN {X 0,Y 157.373,Z 496.877,A -85,B 0,C 180,E1 -23690.933,E2 -23690.933} C_VEL
LIN {X 0,Y 157.318,Z 496.888,A -85,B 0,C 180,E1 -23696.685,E2 -23696.685} C_VEL
LIN {X 0,Y 157.281,Z 496.891,A -85,B 0,C 180,E1 -23702.427,E2 -23702.427} C_VEL
LIN {X 0,Y 157.286,Z 496.891,A -85,B 0,C 180,E1 -23706.457,E2 -23706.457} C_VEL
LIN {X 0,Y 157.216,Z 496.901,A -85,B 0,C 180,E1 -23712.11,E2 -23712.11} C_VEL
LIN {X 0,Y 157.163,Z 496.903,A -85,B 0,C 180,E1 -23717.873,E2 -23717.873} C_VEL
LIN {X 0,Y 157.106,Z 496.913,A -85,B 0,C 180,E1 -23721.223,E2 -23721.223} C_VEL
LIN {X 0,Y 157.015,Z 496.924,A -85,B 0,C 180,E1 -23724.416,E2 -23724.416} C_VEL
LIN {X 0,Y 156.682,Z 496.964,A -85,B 0,C 180,E1 -23728.458,E2 -23728.458} C_VEL
LIN {X 0,Y 156.226,Z 497.112,A -85,B 0,C 180,E1 -23735.602,E2 -23735.602} C_VEL
LIN {X 0,Y 158.367,Z 510.423,A -85,B 0,C 180,E1 -23737.532,E2 -23737.532} C_VEL
LIN {X 0,Y 160.64,Z 523.248,A -85,B 0,C 180,E1 -23739.846,E2 -23739.846} C_VEL
LIN {X 0,Y 159.381,Z 534.477,A -85,B 0,C 180,E1 -23742.352,E2 -23742.352} C_VEL
LIN {X 0,Y 157.924,Z 545.965,A -85,B 0,C 180,E1 -23745.503,E2 -23745.503} C_VEL
LIN {X 0,Y 156.992,Z 554.677,A -85,B 0,C 180,E1 -23748.378,E2 -23748.378} C_VEL
LIN {X 0,Y 156.156,Z 564.37,A -85,B 0,C 180,E1 -23752.24,E2 -23752.24} C_VEL
LIN {X 0,Y 155.685,Z 572.434,A -85,B 0,C 180,E1 -23756.117,E2 -23756.117} C_VEL
LIN {X 0,Y 155.538,Z 579.126,A -85,B 0,C 180,E1 -23760,E2 -23760} C_VEL
LIN {X 0,Y 155.827,Z 584.608,A -85,B 0,C 180,E1 -23763.879,E2 -23763.879} C_VEL
LIN {X 0,Y 156.622,Z 589.966,A -85,B 0,C 180,E1 -23768.496,E2 -23768.496} C_VEL
LIN {X 0,Y 158.293,Z 593.944,A -85,B 0,C 180,E1 -23772.826,E2 -23772.826} C_VEL
LIN {X 0,Y 161.597,Z 597.454,A -85,B 0,C 180,E1 -23777.724,E2 -23777.724} C_VEL
LIN {X 0,Y 166.084,Z 599.704,A -85,B 0,C 180,E1 -23782.386,E2 -23782.386} C_VEL
LIN {X 0,Y 171.924,Z 600.794,A -85,B 0,C 180,E1 -23786.722,E2 -23786.722} C_VEL
LIN {X 0,Y 178.934,Z 600.715,A -85,B 0,C 180,E1 -23790.704,E2 -23790.704} C_VEL
LIN {X 0,Y 186.95,Z 599.507,A -85,B 0,C 180,E1 -23794.325,E2 -23794.325} C_VEL
LIN {X 0,Y 195.971,Z 597.122,A -85,B 0,C 180,E1 -23797.565,E2 -23797.565} C_VEL
LIN {X 0,Y 200.802,Z 595.493,A -85,B 0,C 180,E1 -23799.05,E2 -23799.05} C_VEL
LIN {X 0,Y 204.355,Z 594.188,A -85,B 0,C 180,E1 -23800.834,E2 -23800.834} C_VEL
LIN {X 0,Y 204.262,Z 594.808,A -85,B 0,C 180,E1 -23803.735,E2 -23803.735} C_VEL
LIN {X 0,Y 202.14,Z 596.394,A -85,B 0,C 180,E1 -23805.944,E2 -23805.944} C_VEL
LIN {X 0,Y 198.837,Z 598.405,A -85,B 0,C 180,E1 -23807.812,E2 -23807.812} C_VEL
LIN {X 0,Y 194.385,Z 600.627,A -85,B 0,C 180,E1 -23809.398,E2 -23809.398} C_VEL
LIN {X 0,Y 185.191,Z 604.437,A -85,B 0,C 180,E1 -23812.612,E2 -23812.612} C_VEL
LIN {X 0,Y 177.033,Z 607.18,A -85,B 0,C 180,E1 -23816.235,E2 -23816.235} C_VEL
LIN {X 0,Y 170.079,Z 608.889,A -85,B 0,C 180,E1 -23820.273,E2 -23820.273} C_VEL
LIN {X 0,Y 164.488,Z 609.553,A -85,B 0,C 180,E1 -23824.706,E2 -23824.706} C_VEL
LIN {X 0,Y 160.243,Z 609.172,A -85,B 0,C 180,E1 -23829.459,E2 -23829.459} C_VEL
LIN {X 0,Y 157.527,Z 607.704,A -85,B 0,C 180,E1 -23834.473,E2 -23834.473} C_VEL
LIN {X 0,Y 156.327,Z 605.116,A -85,B 0,C 180,E1 -23839.64,E2 -23839.64} C_VEL
LIN {X 0,Y 156.466,Z 601.271,A -85,B 0,C 180,E1 -23844.846,E2 -23844.846} C_VEL
LIN {X 0,Y 157.222,Z 597.369,A -85,B 0,C 180,E1 -23848.719,E2 -23848.719} C_VEL
LIN {X 0,Y 157.264,Z 593.964,A -85,B 0,C 180,E1 -23851.28,E2 -23851.28} C_VEL
LIN {X 0,Y 157.32,Z 587.742,A -85,B 0,C 180,E1 -23855.126,E2 -23855.126} C_VEL
LIN {X 0,Y 157.426,Z 580.313,A -85,B 0,C 180,E1 -23858.782,E2 -23858.782} C_VEL
LIN {X 0,Y 157.942,Z 572.051,A -85,B 0,C 180,E1 -23862.137,E2 -23862.137} C_VEL
LIN {X 0,Y 158.982,Z 561.294,A -85,B 0,C 180,E1 -23865.709,E2 -23865.709} C_VEL
LIN {X 0,Y 159.431,Z 555.597,A -85,B 0,C 180,E1 -23867.31,E2 -23867.31} C_VEL
LIN {X 0,Y 158.106,Z 544.817,A -85,B 0,C 180,E1 -23869.812,E2 -23869.812} C_VEL
LIN {X 0,Y 156.876,Z 531.321,A -85,B 0,C 180,E1 -23872.383,E2 -23872.383} C_VEL
LIN {X 0,Y 156.246,Z 518.705,A -85,B 0,C 180,E1 -23874.322,E2 -23874.322} C_VEL
LIN {X 0,Y 156.222,Z 509.846,A -85,B 0,C 180,E1 -23875.438,E2 -23875.438} C_VEL
LIN {X 0,Y 157.588,Z 504.758,A -85,B 0,C 180,E1 -23882.355,E2 -23882.355} C_VEL
LIN {X 0,Y 158.359,Z 502.47,A -85,B 0,C 180,E1 -23885.418,E2 -23885.418} C_VEL
LIN {X 0,Y 157.749,Z 501.521,A -85,B 0,C 180,E1 -23886.771,E2 -23886.771} C_VEL
LIN {X 0,Y 154.825,Z 499.997,A -85,B 0,C 180,E1 -23888.887,E2 -23888.887} C_VEL
LIN {X 0,Y 151.702,Z 498.504,A -85,B 0,C 180,E1 -23891.105,E2 -23891.105} C_VEL
LIN {X 0,Y 150.881,Z 497.692,A -85,B 0,C 180,E1 -23892.599,E2 -23892.599} C_VEL
LIN {X 0,Y 150.675,Z 497.716,A -85,B 0,C 180,E1 -23895.601,E2 -23895.601} C_VEL
LIN {X 0,Y 150.275,Z 497.761,A -85,B 0,C 180,E1 -23902.66,E2 -23902.66} C_VEL
LIN {X 0,Y 150.207,Z 497.772,A -85,B 0,C 180,E1 -23909.025,E2 -23909.025} C_VEL
LIN {X 0,Y 150.244,Z 497.766,A -85,B 0,C 180,E1 -23912.718,E2 -23912.718} C_VEL
LIN {X 0,Y 150.353,Z 497.751,A -85,B 0,C 180,E1 -23919.207,E2 -23919.207} C_VEL
LIN {X 0,Y 150.392,Z 497.75,A -85,B 0,C 180,E1 -23923.717,E2 -23923.717} C_VEL
LIN {X 0,Y 150.69,Z 497.708,A -85,B 0,C 180,E1 -23929.249,E2 -23929.249} C_VEL
LIN {X 0,Y 150.764,Z 497.703,A -85,B 0,C 180,E1 -23931.961,E2 -23931.961} C_VEL
LIN {X 0,Y 151.22,Z 497.646,A -85,B 0,C 180,E1 -23940,E2 -23940} C_VEL
LIN {X 0,Y 150.765,Z 497.701,A -85,B 0,C 180,E1 -23948.04,E2 -23948.04} C_VEL
LIN {X 0,Y 150.636,Z 497.72,A -85,B 0,C 180,E1 -23951.546,E2 -23951.546} C_VEL
LIN {X 0,Y 150.369,Z 497.749,A -85,B 0,C 180,E1 -23956.286,E2 -23956.286} C_VEL
LIN {X 0,Y 150.352,Z 497.755,A -85,B 0,C 180,E1 -23960.793,E2 -23960.793} C_VEL
LIN {X 0,Y 150.246,Z 497.768,A -85,B 0,C 180,E1 -23967.283,E2 -23967.283} C_VEL
LIN {X 0,Y 150.217,Z 497.767,A -85,B 0,C 180,E1 -23972.633,E2 -23972.633} C_VEL
LIN {X 0,Y 150.174,Z 497.778,A -85,B 0,C 180,E1 -23977.474,E2 -23977.474} C_VEL
LIN {X 0,Y 150.151,Z 497.775,A -85,B 0,C 180,E1 -23981.505,E2 -23981.505} C_VEL
LIN {X 0,Y 150.127,Z 497.783,A -85,B 0,C 180,E1 -23985.396,E2 -23985.396} C_VEL
LIN {X 0,Y 150.158,Z 497.776,A -85,B 0,C 180,E1 -23989.061,E2 -23989.061} C_VEL
LIN {X 0,Y 150.218,Z 497.772,A -85,B 0,C 180,E1 -23992.69,E2 -23992.69} C_VEL
LIN {X 0,Y 150.221,Z 497.77,A -85,B 0,C 180,E1 -23997.366,E2 -23997.366} C_VEL
LIN {X 0,Y 150.247,Z 497.769,A -85,B 0,C 180,E1 -24002.718,E2 -24002.718} C_VEL
LIN {X 0,Y 150.354,Z 497.751,A -85,B 0,C 180,E1 -24009.208,E2 -24009.208} C_VEL
LIN {X 0,Y 150.365,Z 497.755,A -85,B 0,C 180,E1 -24013.714,E2 -24013.714} C_VEL
LIN {X 0,Y 150.614,Z 497.721,A -85,B 0,C 180,E1 -24019.243,E2 -24019.243} C_VEL
LIN {X 0,Y 150.705,Z 497.714,A -85,B 0,C 180,E1 -24021.958,E2 -24021.958} C_VEL
LIN {X 0,Y 151.221,Z 497.65,A -85,B 0,C 180,E1 -24030,E2 -24030} C_VEL
LIN {X 0,Y 150.709,Z 497.713,A -85,B 0,C 180,E1 -24038.042,E2 -24038.042} C_VEL
LIN {X 0,Y 150.581,Z 497.726,A -85,B 0,C 180,E1 -24041.439,E2 -24041.439} C_VEL
LIN {X 0,Y 150.366,Z 497.755,A -85,B 0,C 180,E1 -24046.287,E2 -24046.287} C_VEL
LIN {X 0,Y 150.354,Z 497.751,A -85,B 0,C 180,E1 -24050.793,E2 -24050.793} C_VEL
LIN {X 0,Y 150.248,Z 497.769,A -85,B 0,C 180,E1 -24057.282,E2 -24057.282} C_VEL
LIN {X 0,Y 150.222,Z 497.77,A -85,B 0,C 180,E1 -24062.634,E2 -24062.634} C_VEL
LIN {X 0,Y 150.214,Z 497.773,A -85,B 0,C 180,E1 -24067.462,E2 -24067.462} C_VEL
LIN {X 0,Y 150.156,Z 497.778,A -85,B 0,C 180,E1 -24071.506,E2 -24071.506} C_VEL
LIN {X 0,Y 150.129,Z 497.784,A -85,B 0,C 180,E1 -24075.395,E2 -24075.395} C_VEL
LIN {X 0,Y 150.098,Z 497.782,A -85,B 0,C 180,E1 -24079.04,E2 -24079.04} C_VEL
LIN {X 0,Y 149.992,Z 497.8,A -85,B 0,C 180,E1 -24082.803,E2 -24082.803} C_VEL
LIN {X 0,Y 149.677,Z 497.835,A -85,B 0,C 180,E1 -24087.692,E2 -24087.692} C_VEL
LIN {X 0,Y 149.213,Z 497.895,A -85,B 0,C 180,E1 -24094.918,E2 -24094.918} C_VEL
LIN {X 0,Y 149.196,Z 498.055,A -85,B 0,C 180,E1 -24095.658,E2 -24095.658} C_VEL
LIN {X 0,Y 151.406,Z 511.655,A -85,B 0,C 180,E1 -24097.754,E2 -24097.754} C_VEL
LIN {X 0,Y 153.462,Z 523.067,A -85,B 0,C 180,E1 -24099.911,E2 -24099.911} C_VEL
LIN {X 0,Y 152.534,Z 531.774,A -85,B 0,C 180,E1 -24101.879,E2 -24101.879} C_VEL
LIN {X 0,Y 151.076,Z 543.658,A -85,B 0,C 180,E1 -24105.175,E2 -24105.175} C_VEL
LIN {X 0,Y 149.986,Z 553.588,A -85,B 0,C 180,E1 -24108.512,E2 -24108.512} C_VEL
LIN {X 0,Y 149.076,Z 564.545,A -85,B 0,C 180,E1 -24113.024,E2 -24113.024} C_VEL
LIN {X 0,Y 148.686,Z 572.956,A -85,B 0,C 180,E1 -24117.29,E2 -24117.29} C_VEL
LIN {X 0,Y 148.617,Z 579.506,A -85,B 0,C 180,E1 -24121.354,E2 -24121.354} C_VEL
LIN {X 0,Y 149.027,Z 585.001,A -85,B 0,C 180,E1 -24125.412,E2 -24125.412} C_VEL
LIN {X 0,Y 150.262,Z 590.835,A -85,B 0,C 180,E1 -24130.782,E2 -24130.782} C_VEL
